# B&R Automation Studio project NAEUL004C00R13L518F00 (part 27)

#### Act_OptP1031TravMask.st
```iecst
ACTION Act_OptP1031TravMask:

	// Interlock Power
	IF p_bTravAxisErr = TRUE AND p_bTravPwrOn = FALSE THEN
		fUIInRtStatOff(ADR(tyP1031MagSetTeach.tyMotionStdTrav.tyBtnPwr.uiMaskRtStat));
		tyP1031MagSetTeach.tyMotionStdTrav.tyBtnPwr.bValue		:= FALSE;
	ELSE
		fUIInRtStatHide(ADR(tyP1031MagSetTeach.tyMotionStdTrav.tyBtnPwr.uiMaskRtStat));
	END_IF

	// Interlock Others Move
	IF p_bTravAxisErr = TRUE OR p_bTravPwrOn = FALSE THEN
		fUIInRtStatOff(ADR(tyP1031MagSetTeach.tyMotionStdTrav.tyBtnOrigin.uiMaskRtStat));
		fUIInRtStatOff(ADR(tyP1031MagSetTeach.tyMotionStdTrav.tyBtnMovRel.uiMaskRtStat));
		fUIInRtStatOff(ADR(tyP1031MagSetTeach.tyMotionStdTrav.tyBtnJogFront.uiMaskRtStat));
		fUIInRtStatOff(ADR(tyP1031MagSetTeach.tyMotionStdTrav.tyBtnJogRear.uiMaskRtStat));
	ELSE
		fUIInRtStatHide(ADR(tyP1031MagSetTeach.tyMotionStdTrav.tyBtnOrigin.uiMaskRtStat));
		fUIInRtStatHide(ADR(tyP1031MagSetTeach.tyMotionStdTrav.tyBtnMovRel.uiMaskRtStat));
		fUIInRtStatHide(ADR(tyP1031MagSetTeach.tyMotionStdTrav.tyBtnJogFront.uiMaskRtStat));
		fUIInRtStatHide(ADR(tyP1031MagSetTeach.tyMotionStdTrav.tyBtnJogRear.uiMaskRtStat));
	END_IF

	// Interlock Move Absolute
	IF p_bTravAxisErr = TRUE OR p_bTravPwrOn = FALSE OR p_bTravIsHomed = FALSE THEN
		fUIInRtStatOff(ADR(tyP1031MagSetTeach.tyTeachTravPosMag1.tyBtn2.uiMaskRtStat));
		fUIInRtStatOff(ADR(tyP1031MagSetTeach.tyTeachTravPosMag2.tyBtn2.uiMaskRtStat));
		fUIInRtStatOff(ADR(tyP1031MagSetTeach.tyTeachTravPosMag3.tyBtn2.uiMaskRtStat));
		fUIInRtStatOff(ADR(tyP1031MagSetTeach.tyMotionStdTrav.tyBtnMovAbs.uiMaskRtStat));
	ELSE
		fUIInRtStatHide(ADR(tyP1031MagSetTeach.tyTeachTravPosMag1.tyBtn2.uiMaskRtStat));
		fUIInRtStatHide(ADR(tyP1031MagSetTeach.tyTeachTravPosMag2.tyBtn2.uiMaskRtStat));
		fUIInRtStatHide(ADR(tyP1031MagSetTeach.tyTeachTravPosMag3.tyBtn2.uiMaskRtStat));
		fUIInRtStatHide(ADR(tyP1031MagSetTeach.tyMotionStdTrav.tyBtnMovAbs.uiMaskRtStat));
	END_IF

	//Interlock Limit Sensor
	IF tyP1031MagSetTeach.tyMotionStdTrav.tyBtnRearLmtSen.bValue = TRUE THEN
		fUIInRtStatOff(ADR(tyP1031MagSetTeach.tyMotionStdTrav.tyBtnJogRear.uiMaskRtStat));
	END_IF

	IF tyP1031MagSetTeach.tyMotionStdTrav.tyBtnFrontLmtSen.bValue = TRUE THEN
		fUIInRtStatOff(ADR(tyP1031MagSetTeach.tyMotionStdTrav.tyBtnJogFront.uiMaskRtStat));
	END_IF

	// Interlock When Moving
	IF tyP1031MagSetTeach.tyMotionStdTrav.tyBtnOrigin.bRtCompl = TRUE THEN
		fUIInRtStatOff(ADR(tyP1031MagSetTeach.tyMotionStdTrav.tyBtnMovAbs.uiMaskRtStat));
		fUIInRtStatOff(ADR(tyP1031MagSetTeach.tyMotionStdTrav.tyBtnMovRel.uiMaskRtStat));
		fUIInRtStatOff(ADR(tyP1031MagSetTeach.tyMotionStdTrav.tyBtnJogFront.uiMaskRtStat));
		fUIInRtStatOff(ADR(tyP1031MagSetTeach.tyMotionStdTrav.tyBtnJogRear.uiMaskRtStat));

		fUIInRtStatOff(ADR(tyP1031MagSetTeach.tyTeachTravPosMag1.tyBtn2.uiMaskRtStat));
		fUIInRtStatOff(ADR(tyP1031MagSetTeach.tyTeachTravPosMag2.tyBtn2.uiMaskRtStat));
		fUIInRtStatOff(ADR(tyP1031MagSetTeach.tyTeachTravPosMag3.tyBtn2.uiMaskRtStat));

	ELSIF tyP1031MagSetTeach.tyMotionStdTrav.tyBtnMovAbs.bRtCompl = TRUE THEN
		fUIInRtStatOff(ADR(tyP1031MagSetTeach.tyMotionStdTrav.tyBtnOrigin.uiMaskRtStat));
		fUIInRtStatOff(ADR(tyP1031MagSetTeach.tyMotionStdTrav.tyBtnMovRel.uiMaskRtStat));
		fUIInRtStatOff(ADR(tyP1031MagSetTeach.tyMotionStdTrav.tyBtnJogFront.uiMaskRtStat));
		fUIInRtStatOff(ADR(tyP1031MagSetTeach.tyMotionStdTrav.tyBtnJogRear.uiMaskRtStat));

		fUIInRtStatOff(ADR(tyP1031MagSetTeach.tyTeachTravPosMag1.tyBtn2.uiMaskRtStat));
		fUIInRtStatOff(ADR(tyP1031MagSetTeach.tyTeachTravPosMag2.tyBtn2.uiMaskRtStat));
		fUIInRtStatOff(ADR(tyP1031MagSetTeach.tyTeachTravPosMag3.tyBtn2.uiMaskRtStat));

	ELSIF tyP1031MagSetTeach.tyMotionStdTrav.tyBtnMovRel.bRtCompl = TRUE THEN
		fUIInRtStatOff(ADR(tyP1031MagSetTeach.tyMotionStdTrav.tyBtnOrigin.uiMaskRtStat));
		fUIInRtStatOff(ADR(tyP1031MagSetTeach.tyMotionStdTrav.tyBtnMovAbs.uiMaskRtStat));
		fUIInRtStatOff(ADR(tyP1031MagSetTeach.tyMotionStdTrav.tyBtnJogFront.uiMaskRtStat));
		fUIInRtStatOff(ADR(tyP1031MagSetTeach.tyMotionStdTrav.tyBtnJogRear.uiMaskRtStat));

		fUIInRtStatOff(ADR(tyP1031MagSetTeach.tyTeachTravPosMag1.tyBtn2.uiMaskRtStat));
		fUIInRtStatOff(ADR(tyP1031MagSetTeach.tyTeachTravPosMag2.tyBtn2.uiMaskRtStat));
		fUIInRtStatOff(ADR(tyP1031MagSetTeach.tyTeachTravPosMag3.tyBtn2.uiMaskRtStat));

	ELSIF tyP1031MagSetTeach.tyMotionStdTrav.tyBtnJogRear.bRtCompl = TRUE OR tyP1031MagSetTeach.tyMotionStdTrav.tyBtnJogRear.bValue = TRUE THEN
		fUIInRtStatOff(ADR(tyP1031MagSetTeach.tyMotionStdTrav.tyBtnOrigin.uiMaskRtStat));
		fUIInRtStatOff(ADR(tyP1031MagSetTeach.tyMotionStdTrav.tyBtnMovAbs.uiMaskRtStat));
		fUIInRtStatOff(ADR(tyP1031MagSetTeach.tyMotionStdTrav.tyBtnMovRel.uiMaskRtStat));
		fUIInRtStatOff(ADR(tyP1031MagSetTeach.tyMotionStdTrav.tyBtnJogFront.uiMaskRtStat));

		fUIInRtStatOff(ADR(tyP1031MagSetTeach.tyTeachTravPosMag1.tyBtn2.uiMaskRtStat));
		fUIInRtStatOff(ADR(tyP1031MagSetTeach.tyTeachTravPosMag2.tyBtn2.uiMaskRtStat));
		fUIInRtStatOff(ADR(tyP1031MagSetTeach.tyTeachTravPosMag3.tyBtn2.uiMaskRtStat));

	ELSIF tyP1031MagSetTeach.tyMotionStdTrav.tyBtnJogFront.bRtCompl = TRUE OR tyP1031MagSetTeach.tyMotionStdTrav.tyBtnJogFront.bValue = TRUE THEN
		fUIInRtStatOff(ADR(tyP1031MagSetTeach.tyMotionStdTrav.tyBtnOrigin.uiMaskRtStat));
		fUIInRtStatOff(ADR(tyP1031MagSetTeach.tyMotionStdTrav.tyBtnMovAbs.uiMaskRtStat));
		fUIInRtStatOff(ADR(tyP1031MagSetTeach.tyMotionStdTrav.tyBtnMovRel.uiMaskRtStat));
		fUIInRtStatOff(ADR(tyP1031MagSetTeach.tyMotionStdTrav.tyBtnJogRear.uiMaskRtStat));

		fUIInRtStatOff(ADR(tyP1031MagSetTeach.tyTeachTravPosMag1.tyBtn2.uiMaskRtStat));
		fUIInRtStatOff(ADR(tyP1031MagSetTeach.tyTeachTravPosMag2.tyBtn2.uiMaskRtStat));
		fUIInRtStatOff(ADR(tyP1031MagSetTeach.tyTeachTravPosMag3.tyBtn2.uiMaskRtStat));

	ELSIF tyP1031MagSetTeach.tyTeachTravPosMag1.tyBtn2.bRtCompl = TRUE THEN
		fUIInRtStatOff(ADR(tyP1031MagSetTeach.tyMotionStdTrav.tyBtnOrigin.uiMaskRtStat));
		fUIInRtStatOff(ADR(tyP1031MagSetTeach.tyMotionStdTrav.tyBtnMovAbs.uiMaskRtStat));
		fUIInRtStatOff(ADR(tyP1031MagSetTeach.tyMotionStdTrav.tyBtnMovRel.uiMaskRtStat));
		fUIInRtStatOff(ADR(tyP1031MagSetTeach.tyMotionStdTrav.tyBtnJogFront.uiMaskRtStat));
		fUIInRtStatOff(ADR(tyP1031MagSetTeach.tyMotionStdTrav.tyBtnJogRear.uiMaskRtStat));

	ELSIF tyP1031MagSetTeach.tyTeachTravPosMag2.tyBtn2.bRtCompl = TRUE THEN
		fUIInRtStatOff(ADR(tyP1031MagSetTeach.tyMotionStdTrav.tyBtnOrigin.uiMaskRtStat));
		fUIInRtStatOff(ADR(tyP1031MagSetTeach.tyMotionStdTrav.tyBtnMovAbs.uiMaskRtStat));
		fUIInRtStatOff(ADR(tyP1031MagSetTeach.tyMotionStdTrav.tyBtnMovRel.uiMaskRtStat));
		fUIInRtStatOff(ADR(tyP1031MagSetTeach.tyMotionStdTrav.tyBtnJogFront.uiMaskRtStat));
		fUIInRtStatOff(ADR(tyP1031MagSetTeach.tyMotionStdTrav.tyBtnJogRear.uiMaskRtStat));

	ELSIF tyP1031MagSetTeach.tyTeachTravPosMag3.tyBtn2.bRtCompl = TRUE THEN
		fUIInRtStatOff(ADR(tyP1031MagSetTeach.tyMotionStdTrav.tyBtnOrigin.uiMaskRtStat));
		fUIInRtStatOff(ADR(tyP1031MagSetTeach.tyMotionStdTrav.tyBtnMovAbs.uiMaskRtStat));
		fUIInRtStatOff(ADR(tyP1031MagSetTeach.tyMotionStdTrav.tyBtnMovRel.uiMaskRtStat));
		fUIInRtStatOff(ADR(tyP1031MagSetTeach.tyMotionStdTrav.tyBtnJogFront.uiMaskRtStat));
		fUIInRtStatOff(ADR(tyP1031MagSetTeach.tyMotionStdTrav.tyBtnJogRear.uiMaskRtStat));

	END_IF

	//Axis Error
	IF tyP1031MagSetTeach.tyMotionStdTrav.tyBtnPwr.bRtCompl = TRUE  THEN
		fUIInRtStatOff(ADR(tyP1031MagSetTeach.tyMotionStdTrav.tyBtnRst.uiMaskRtStat));
	ELSE
		fUIInRtStatHide(ADR(tyP1031MagSetTeach.tyMotionStdTrav.tyBtnRst.uiMaskRtStat));
	END_IF

	//Interlock Button Get
	IF p_bTravAxisErr = TRUE OR p_bTravIsHomed = FALSE OR p_bTravFwdLmtSen = TRUE OR p_bTravRevLmtSen = TRUE THEN
		fUIInRtStatOff(ADR(tyP1031MagSetTeach.tyTeachTravPosMag1.tyBtn1.uiMaskRtStat));
		fUIInRtStatOff(ADR(tyP1031MagSetTeach.tyTeachTravPosMag2.tyBtn1.uiMaskRtStat));
		fUIInRtStatOff(ADR(tyP1031MagSetTeach.tyTeachTravPosMag3.tyBtn1.uiMaskRtStat));
	ELSE
		fUIInRtStatHide(ADR(tyP1031MagSetTeach.tyTeachTravPosMag1.tyBtn1.uiMaskRtStat));
		fUIInRtStatHide(ADR(tyP1031MagSetTeach.tyTeachTravPosMag2.tyBtn1.uiMaskRtStat));
		fUIInRtStatHide(ADR(tyP1031MagSetTeach.tyTeachTravPosMag3.tyBtn1.uiMaskRtStat));
	END_IF

END_ACTION
```

#### Act_OptP1031TravUpdtDat.st
```iecst
ACTION Act_OptP1031TravUpdtDat:

	tyP1031MagSetTeach.tyMotionStdTrav.tyNumCurrPos.diValue			:= p_diTravActualPos;
	tyP1031MagSetTeach.tyMotionStdTrav.tyNumErrCode.diValue			:= UDINT_TO_DINT(p_udiTravAxisErrID);
	tyP1031MagSetTeach.tyMotionStdTrav.tyBitmapPwr.usiValueIdx		:= BOOL_TO_USINT(p_bTravPwrOn);
	tyP1031MagSetTeach.tyMotionStdTrav.tyBitmapRst.usiValueIdx		:= BOOL_TO_USINT(NOT p_bTravAxisErr);
	tyP1031MagSetTeach.tyMotionStdTrav.tyBitmapOrigin.usiValueIdx	:= BOOL_TO_USINT(p_bTravIsHomed);
	tyP1031MagSetTeach.tyMotionStdTrav.tyBtnFrontLmtSen.bValue		:= p_bTravFrontSen;
	tyP1031MagSetTeach.tyMotionStdTrav.tyBtnRearLmtSen.bValue		:= p_bTravRearSen;

	//Machine Bitmap
	IF p_bTravIsHomed = TRUE THEN
		IF p_diTravActualPos <= (p_tyNtParamCurr.tyUITravTargetPos.diMax / 3) THEN
			tyP1031MagSetTeach.tyMotionStdTrav.tyBitmapMc.uiValueIdx 	:= 5;
		ELSIF p_diTravActualPos <= (p_tyNtParamCurr.tyUITravTargetPos.diMax / 3 * 2) THEN
			tyP1031MagSetTeach.tyMotionStdTrav.tyBitmapMc.uiValueIdx 	:= 6;
		ELSE
			tyP1031MagSetTeach.tyMotionStdTrav.tyBitmapMc.uiValueIdx 	:= 7;
		END_IF
	ELSE
		tyP1031MagSetTeach.tyMotionStdTrav.tyBitmapMc.uiValueIdx	:= 5;
	END_IF

	IF p_tyNtParamCurr.eProjMag = ULMagDual THEN
		IF p_tyNtParamCurr.bProjLifterMagPlatform AND p_tyNtParamCurr.bUIConvDirRL THEN
			IF 	tyP1031MagSetTeach.tyMotionStdTrav.tyBitmapMc.uiValueIdx < 700 THEN
				tyP1031MagSetTeach.tyMotionStdTrav.tyBitmapMc.uiValueIdx	:= tyP1031MagSetTeach.tyMotionStdTrav.tyBitmapMc.uiValueIdx + 700;
			END_IF
		ELSIF p_tyNtParamCurr.bProjLifterMagPlatform THEN
			IF 	tyP1031MagSetTeach.tyMotionStdTrav.tyBitmapMc.uiValueIdx < 600 THEN
				tyP1031MagSetTeach.tyMotionStdTrav.tyBitmapMc.uiValueIdx	:= tyP1031MagSetTeach.tyMotionStdTrav.tyBitmapMc.uiValueIdx + 600;
			END_IF
		ELSIF p_tyNtParamCurr.bMagAutoVerifyPrep = FALSE THEN
			IF 	tyP1031MagSetTeach.tyMotionStdTrav.tyBitmapMc.uiValueIdx < 100 THEN
				tyP1031MagSetTeach.tyMotionStdTrav.tyBitmapMc.uiValueIdx	:= tyP1031MagSetTeach.tyMotionStdTrav.tyBitmapMc.uiValueIdx + 300;
			END_IF
		ELSE
			IF 	tyP1031MagSetTeach.tyMotionStdTrav.tyBitmapMc.uiValueIdx < 300 THEN
				tyP1031MagSetTeach.tyMotionStdTrav.tyBitmapMc.uiValueIdx	:= tyP1031MagSetTeach.tyMotionStdTrav.tyBitmapMc.uiValueIdx + 300;
			END_IF
		END_IF
	ELSIF p_tyNtParamCurr.eProjMag = ULMagTriple THEN
		IF p_tyNtParamCurr.bProjLifterMagPlatform AND p_tyNtParamCurr.bUIConvDirRL THEN
			IF 	tyP1031MagSetTeach.tyMotionStdTrav.tyBitmapMc.uiValueIdx < 800 THEN
				tyP1031MagSetTeach.tyMotionStdTrav.tyBitmapMc.uiValueIdx	:= tyP1031MagSetTeach.tyMotionStdTrav.tyBitmapMc.uiValueIdx + 800;
			END_IF
		ELSIF p_tyNtParamCurr.bProjLifterMagPlatform THEN
			IF 	tyP1031MagSetTeach.tyMotionStdTrav.tyBitmapMc.uiValueIdx < 500 THEN
				tyP1031MagSetTeach.tyMotionStdTrav.tyBitmapMc.uiValueIdx	:= tyP1031MagSetTeach.tyMotionStdTrav.tyBitmapMc.uiValueIdx + 500;
			END_IF
		ELSIF p_tyNtParamCurr.bMagAutoVerifyPrep = TRUE AND p_tyNtParamCurr.bProjMotorizedPusherPrep = FALSE THEN
			IF 	tyP1031MagSetTeach.tyMotionStdTrav.tyBitmapMc.uiValueIdx < 200 THEN
				tyP1031MagSetTeach.tyMotionStdTrav.tyBitmapMc.uiValueIdx	:= tyP1031MagSetTeach.tyMotionStdTrav.tyBitmapMc.uiValueIdx + 200;
			END_IF
		ELSIF p_tyNtParamCurr.bMagAutoVerifyPrep = FALSE AND p_tyNtParamCurr.bProjMotorizedPusherPrep = TRUE THEN
			IF 	tyP1031MagSetTeach.tyMotionStdTrav.tyBitmapMc.uiValueIdx < 400 THEN
				tyP1031MagSetTeach.tyMotionStdTrav.tyBitmapMc.uiValueIdx	:= tyP1031MagSetTeach.tyMotionStdTrav.tyBitmapMc.uiValueIdx + 400;
			END_IF
		END_IF
	END_IF

END_ACTION
```

#### Act_OptP1031TravKeypad.st
```iecst
ACTION Act_OptP1031TravKeypad:

	IF fUIOutRtStatTPIsOpen(ADR(tyP1031MagSetTeach.tyMotionStdTrav.tyNumTargetPos.uiRtStat)) = TRUE THEN
		tyProperty.tyKeypad.tyStringTitle.sKeypadTitle		:= tyP1031MagSetTeach.tyMotionStdTrav.tyNumTargetPos.sKeypadTitle;

	ELSIF fUIOutRtStatTPIsOpen(ADR(tyP1031MagSetTeach.tyMotionStdTrav.tyNumStepSize.uiRtStat)) = TRUE THEN
		tyProperty.tyKeypad.tyStringTitle.sKeypadTitle		:= tyP1031MagSetTeach.tyMotionStdTrav.tyNumStepSize.sKeypadTitle;

	ELSIF fUIOutRtStatTPIsOpen(ADR(tyP1031MagSetTeach.tyMotionStdTrav.tyNumNomSpd.uiRtStat)) = TRUE THEN
		tyProperty.tyKeypad.tyStringTitle.sKeypadTitle		:= tyP1031MagSetTeach.tyMotionStdTrav.tyNumNomSpd.sKeypadTitle;

	ELSIF fUIOutRtStatTPIsOpen(ADR(tyP1031MagSetTeach.tyMotionStdTrav.tyNumSlwSpd.uiRtStat)) = TRUE THEN
		tyProperty.tyKeypad.tyStringTitle.sKeypadTitle		:= tyP1031MagSetTeach.tyMotionStdTrav.tyNumSlwSpd.sKeypadTitle;
	END_IF

END_ACTION
```

#### Act_OptP1031TravRstMnl.st
```iecst
ACTION Act_OptP1031TravRstMnl:

	IF EDGEPOS((bManualMod = FALSE) OR (p_eTravStatus = Error)) THEN

		bJogSlow				:= FALSE;
		bJogFast				:= FALSE;
		fbJogSlowToFastDlyTm.IN	:= FALSE;

		tyP1031MagSetTeach.tyMotionStdTrav.tyBtnPwr.bRtCompl			:= FALSE;
		tyP1031MagSetTeach.tyMotionStdTrav.tyBtnStop.bRtCompl			:= FALSE;
		tyP1031MagSetTeach.tyMotionStdTrav.tyBtnOrigin.bRtCompl			:= FALSE;
		tyP1031MagSetTeach.tyMotionStdTrav.tyBtnRst.bRtCompl			:= FALSE;
		tyP1031MagSetTeach.tyMotionStdTrav.tyBtnMovAbs.bRtCompl			:= FALSE;
		tyP1031MagSetTeach.tyMotionStdTrav.tyBtnMovRel.bRtCompl			:= FALSE;
		tyP1031MagSetTeach.tyMotionStdTrav.tyBtnJogFront.bRtCompl		:= FALSE;
		tyP1031MagSetTeach.tyMotionStdTrav.tyBtnJogRear.bRtCompl		:= FALSE;

		tyP1031MagSetTeach.tyTeachTravPosMag1.tyBtn2.bRtCompl			:= FALSE;
		tyP1031MagSetTeach.tyTeachTravPosMag2.tyBtn2.bRtCompl			:= FALSE;
		tyP1031MagSetTeach.tyTeachTravPosMag3.tyBtn2.bRtCompl			:= FALSE;

		tyP1031MagSetTeach.tyMotionStdTrav.tyBtnPwr.bValue				:= FALSE;
		tyP1031MagSetTeach.tyMotionStdTrav.tyBtnStop.bValue				:= TRUE;
		tyP1031MagSetTeach.tyMotionStdTrav.tyBtnOrigin.bValue			:= FALSE;
		tyP1031MagSetTeach.tyMotionStdTrav.tyBtnRst.bValue				:= FALSE;
		tyP1031MagSetTeach.tyMotionStdTrav.tyBtnMovAbs.bValue			:= FALSE;
		tyP1031MagSetTeach.tyMotionStdTrav.tyBtnMovRel.bValue			:= FALSE;
		tyP1031MagSetTeach.tyMotionStdTrav.tyBtnJogFront.bValue			:= FALSE;
		tyP1031MagSetTeach.tyMotionStdTrav.tyBtnJogRear.bValue			:= FALSE;

		tyP1031MagSetTeach.tyTeachTravPosMag1.tyBtn2.bValue				:= FALSE;
		tyP1031MagSetTeach.tyTeachTravPosMag2.tyBtn2.bValue				:= FALSE;
		tyP1031MagSetTeach.tyTeachTravPosMag3.tyBtn2.bValue				:= FALSE;

		tyP1031MagSetTeach.tyMotionStdTrav.tyBtnPwr.bRtLk				:= FALSE;
		tyP1031MagSetTeach.tyMotionStdTrav.tyBtnStop.bRtLk				:= TRUE;
		tyP1031MagSetTeach.tyMotionStdTrav.tyBtnOrigin.bRtLk			:= FALSE;
		tyP1031MagSetTeach.tyMotionStdTrav.tyBtnRst.bRtLk				:= FALSE;
		tyP1031MagSetTeach.tyMotionStdTrav.tyBtnMovAbs.bRtLk			:= FALSE;
		tyP1031MagSetTeach.tyMotionStdTrav.tyBtnMovRel.bRtLk			:= FALSE;
		tyP1031MagSetTeach.tyMotionStdTrav.tyBtnJogFront.bRtLk			:= FALSE;
		tyP1031MagSetTeach.tyMotionStdTrav.tyBtnJogRear.bRtLk			:= FALSE;

		tyP1031MagSetTeach.tyTeachTravPosMag1.tyBtn2.bRtLk				:= FALSE;
		tyP1031MagSetTeach.tyTeachTravPosMag2.tyBtn2.bRtLk				:= FALSE;
		tyP1031MagSetTeach.tyTeachTravPosMag3.tyBtn2.bRtLk				:= FALSE;

		tyP1031MagSetTeach.tyMotionStdTrav.tyBtnPwr.uiMaskRtStat		:= TRUE;
		tyP1031MagSetTeach.tyMotionStdTrav.tyBtnOrigin.uiMaskRtStat		:= FALSE;
		tyP1031MagSetTeach.tyMotionStdTrav.tyBtnRst.uiMaskRtStat		:= TRUE;
		tyP1031MagSetTeach.tyMotionStdTrav.tyBtnMovAbs.uiMaskRtStat		:= FALSE;
		tyP1031MagSetTeach.tyMotionStdTrav.tyBtnMovRel.uiMaskRtStat		:= FALSE;
		tyP1031MagSetTeach.tyMotionStdTrav.tyBtnJogFront.uiMaskRtStat	:= FALSE;
		tyP1031MagSetTeach.tyMotionStdTrav.tyBtnJogRear.uiMaskRtStat	:= FALSE;

		tyP1031MagSetTeach.tyTeachTravPosMag1.tyBtn2.uiMaskRtStat		:= FALSE;
		tyP1031MagSetTeach.tyTeachTravPosMag2.tyBtn2.uiMaskRtStat		:= FALSE;
		tyP1031MagSetTeach.tyTeachTravPosMag3.tyBtn2.uiMaskRtStat		:= FALSE;

		eInShutterAct	:= PneuActIdle;
		eOutShutterAct	:= PneuActIdle;
		eOutShutterAct2	:= PneuActIdle;
		eOutShutterAct3	:= PneuActIdle;
		eTravAct	:= TravActIdle;

		tyP1031MagSetTeach.tyInOutletShutterFB.tyBtnClose.bRtCompl	:= FALSE;
		tyP1031MagSetTeach.tyInOutletShutterFB.tyBtnClose.bValue	:= FALSE;
		tyP1031MagSetTeach.tyInOutletShutterFB.tyBtnOpen.bRtCompl	:= FALSE;
		tyP1031MagSetTeach.tyInOutletShutterFB.tyBtnOpen.bValue	:= FALSE;

	END_IF

END_ACTION
```

#### Act_OptP1031LifterTeach.st
```iecst
ACTION Act_OptP1031LifterTeach:

	IF tyP1031MagSetTeach.tyTeachLifterMag1Slt1Pos.tyBtn1.bRtCompl = TRUE THEN // Teach Lifter Magazine 1 Slot 1 Position

		p_tyC0008MsgBox ACCESS ADR(tyP1031MagSetTeach.tyMsgBoxUpdtLifterMag1Slt1Pos);

		IF tyP1031MagSetTeach.tyMsgBoxUpdtLifterMag1Slt1Pos.tyBtnNo.bRtCompl THEN
			tyP1031MagSetTeach.tyMsgBoxUpdtLifterMag1Slt1Pos.tyBtnNo.bRtCompl 	:= FALSE;
			tyP1031MagSetTeach.tyMsgBoxUpdtLifterMag1Slt1Pos.tyBtnNo.bValue 	:= FALSE;

			p_tyC0008MsgBox ACCESS ADR(tyP1031MagSetTeach.tyMsgBoxHide);

			//Write Actual Position To Magazine Setting.
			tyP1030MagSet.tyMagSet.tyNumLifterMag1Slt1Pos.diValue 	:= p_diLifterBtmActualPos;
			tyP1030MagSet.tyMagSet.tyNumLifterMag1Slt1Pos.bRtCompl	:= TRUE;

			//Back To Magazine Settings
			eChgPage	:= UIP1030MagSet;

			fUIInRtStatHide(ADR(tyP1030MagSet.tyMagSet.tyBtnSave.uiMaskRtStat));

			tyP1031MagSetTeach.tyTeachLifterMag1Slt1Pos.tyBtn1.bRtCompl	:= FALSE;
			tyP1031MagSetTeach.tyTeachLifterMag1Slt1Pos.tyBtn1.bValue	:= FALSE;

		END_IF

	ELSIF tyP1031MagSetTeach.tyTeachLifterMag2Slt1Pos.tyBtn1.bRtCompl = TRUE THEN // Teach Lifter Magazine 2 Slot 1 Position

		p_tyC0008MsgBox ACCESS ADR(tyP1031MagSetTeach.tyMsgBoxUpdtLifterMag2Slt1Pos);

		IF tyP1031MagSetTeach.tyMsgBoxUpdtLifterMag2Slt1Pos.tyBtnNo.bRtCompl THEN
			tyP1031MagSetTeach.tyMsgBoxUpdtLifterMag2Slt1Pos.tyBtnNo.bRtCompl 	:= FALSE;
			tyP1031MagSetTeach.tyMsgBoxUpdtLifterMag2Slt1Pos.tyBtnNo.bValue 	:= FALSE;

			p_tyC0008MsgBox ACCESS ADR(tyP1031MagSetTeach.tyMsgBoxHide);

			IF p_tyNtParamCurr.bProjMagConvLane2Prep THEN
				tyP1030MagSet.tyMagSet.tyNumLifterMag2Slt1Pos.diValue 	:= p_diLifter2ActualPos;
			ELSE
				//Write Actual Position To Magazine Setting.
				tyP1030MagSet.tyMagSet.tyNumLifterMag2Slt1Pos.diValue 	:= p_diLifterBtmActualPos;
			END_IF

			tyP1030MagSet.tyMagSet.tyNumLifterMag2Slt1Pos.bRtCompl	:= TRUE;

			//Back To Magazine Settings
			eChgPage	:= UIP1030MagSet;

			fUIInRtStatHide(ADR(tyP1030MagSet.tyMagSet.tyBtnSave.uiMaskRtStat));

			tyP1031MagSetTeach.tyTeachLifterMag2Slt1Pos.tyBtn1.bRtCompl	:= FALSE;
			tyP1031MagSetTeach.tyTeachLifterMag2Slt1Pos.tyBtn1.bValue	:= FALSE;

		END_IF

	ELSIF tyP1031MagSetTeach.tyTeachLifterMag3Slt1Pos.tyBtn1.bRtCompl = TRUE THEN // Teach Lifter Magazine 3 Slot 1 Position

		p_tyC0008MsgBox ACCESS ADR(tyP1031MagSetTeach.tyMsgBoxUpdtLifterMag3Slt1Pos);

		IF tyP1031MagSetTeach.tyMsgBoxUpdtLifterMag3Slt1Pos.tyBtnNo.bRtCompl THEN
			tyP1031MagSetTeach.tyMsgBoxUpdtLifterMag3Slt1Pos.tyBtnNo.bRtCompl 	:= FALSE;
			tyP1031MagSetTeach.tyMsgBoxUpdtLifterMag3Slt1Pos.tyBtnNo.bValue 	:= FALSE;

			p_tyC0008MsgBox ACCESS ADR(tyP1031MagSetTeach.tyMsgBoxHide);

			//Write Actual Position To Magazine Setting.
			tyP1030MagSet.tyMagSet.tyNumLifterMag3Slt1Pos.diValue 	:= p_diLifterBtmActualPos;
			tyP1030MagSet.tyMagSet.tyNumLifterMag3Slt1Pos.bRtCompl	:= TRUE;

			//Back To Magazine Settings
			eChgPage	:= UIP1030MagSet;

			fUIInRtStatHide(ADR(tyP1030MagSet.tyMagSet.tyBtnSave.uiMaskRtStat));

			tyP1031MagSetTeach.tyTeachLifterMag3Slt1Pos.tyBtn1.bRtCompl	:= FALSE;
			tyP1031MagSetTeach.tyTeachLifterMag3Slt1Pos.tyBtn1.bValue	:= FALSE;

		END_IF

	END_IF

END_ACTION
```

#### Act_OptP1031LifterFBCtrl.st
```iecst
ACTION Act_OptP1031LifterFBCtrl:

	fbJogSlowToFastDlyTm.PT	:= T#2s;
	fbJogSlowToFastDlyTm;
	fbLmtRstTm;

	//Lifter Safety Sensor Interruption
	IF EDGENEG(p_tyDI.bLifterSafetyLmtSW1 AND p_tyDI.bLifterSafetyLmtSW2 AND p_tyDI.bLifterTimingBeltSen) THEN
		tyP1031MagSetTeach.tyMotionStdLifter.tyBtnStop.bRtCompl	:= TRUE;
	END_IF

//	IF EDGEPOS((p_udiLifterBtmAxisErrID = 21570 OR p_udiLifterBtmAxisErrID = 21571) AND tyP1031MagSetTeach.tyMotionStdLifter.tyBtnJogDown.bValue = FALSE AND tyP1031MagSetTeach.tyMotionStdLifter.tyBtnJogUp.bValue = FALSE) THEN
	IF EDGEPOS((p_bLifterBtmFwdLmtSen OR p_bLifterBtmRevLmtSen OR p_udiLifterBtmAxisErrID = 21570 OR p_udiLifterBtmAxisErrID = 21571)
		AND tyP1026McSetTeach.tyMotionStdLifter.tyBtnJogDown.bValue = FALSE
		AND tyP1026McSetTeach.tyMotionStdLifter.tyBtnJogUp.bValue = FALSE) THEN
			fbLmtRstTm.IN				:= TRUE;
	END_IF

	IF fbLmtRstTm.Q = TRUE THEN
		tyP1031MagSetTeach.tyMotionStdLifter.tyBtnRst.bRtCompl		:= TRUE;
	END_IF

	IF (tyP1031MagSetTeach.tyMotionStdLifter.tyBtnJogUp.bValue = FALSE AND tyP1031MagSetTeach.tyMotionStdLifter.tyBtnJogDown.bValue = FALSE) AND (p_bLifterBtmJogging = TRUE) THEN
		bJogStopLifter	:= TRUE;
	END_IF

	IF tyP1031MagSetTeach.tyMotionStdLifter.tyBtnStop.bRtCompl = TRUE THEN
		eLifterBtmAct		:= LifterActStop;

		IF p_eLifterBtmStat = LifterActStop AND p_eLifterBtmStatus = Done THEN
			eLifterBtmAct	:= LifterActIdle;

			tyP1031MagSetTeach.tyMotionStdLifter.tyBtnStop.bRtCompl			:= FALSE;
			tyP1031MagSetTeach.tyMotionStdLifter.tyBtnJogDown.bRtCompl		:= FALSE;
			tyP1031MagSetTeach.tyMotionStdLifter.tyBtnJogUp.bRtCompl		:= FALSE;
			tyP1031MagSetTeach.tyMotionStdLifter.tyBtnOrigin.bRtCompl		:= FALSE;
			tyP1031MagSetTeach.tyMotionStdLifter.tyBtnMovAbs.bRtCompl		:= FALSE;
			tyP1031MagSetTeach.tyMotionStdLifter.tyBtnMovRel.bRtCompl		:= FALSE;

			tyP1031MagSetTeach.tyTeachLifterMag1Slt1Pos.tyBtn2.bRtCompl		:= FALSE;
			tyP1031MagSetTeach.tyTeachLifterMag2Slt1Pos.tyBtn2.bRtCompl		:= FALSE;
			tyP1031MagSetTeach.tyTeachLifterMag3Slt1Pos.tyBtn2.bRtCompl		:= FALSE;

			tyP1031MagSetTeach.tyMotionStdLifter.tyBtnStop.bValue			:= TRUE;
			tyP1031MagSetTeach.tyMotionStdLifter.tyBtnJogDown.bValue		:= FALSE;
			tyP1031MagSetTeach.tyMotionStdLifter.tyBtnJogUp.bValue			:= FALSE;
			tyP1031MagSetTeach.tyMotionStdLifter.tyBtnOrigin.bValue			:= FALSE;
			tyP1031MagSetTeach.tyMotionStdLifter.tyBtnMovAbs.bValue			:= FALSE;
			tyP1031MagSetTeach.tyMotionStdLifter.tyBtnMovRel.bValue			:= FALSE;

			tyP1031MagSetTeach.tyTeachLifterMag1Slt1Pos.tyBtn2.bValue		:= FALSE;
			tyP1031MagSetTeach.tyTeachLifterMag2Slt1Pos.tyBtn2.bValue		:= FALSE;
			tyP1031MagSetTeach.tyTeachLifterMag3Slt1Pos.tyBtn2.bValue		:= FALSE;

			tyP1031MagSetTeach.tyMotionStdLifter.tyBtnStop.bRtLk			:= TRUE;
			tyP1031MagSetTeach.tyMotionStdLifter.tyBtnJogDown.bRtLk			:= FALSE;
			tyP1031MagSetTeach.tyMotionStdLifter.tyBtnJogUp.bRtLk			:= FALSE;
			tyP1031MagSetTeach.tyMotionStdLifter.tyBtnOrigin.bRtLk			:= FALSE;
			tyP1031MagSetTeach.tyMotionStdLifter.tyBtnMovAbs.bRtLk			:= FALSE;
			tyP1031MagSetTeach.tyMotionStdLifter.tyBtnMovRel.bRtLk			:= FALSE;

			tyP1031MagSetTeach.tyTeachLifterMag1Slt1Pos.tyBtn2.bRtLk		:= FALSE;
			tyP1031MagSetTeach.tyTeachLifterMag2Slt1Pos.tyBtn2.bRtLk		:= FALSE;
			tyP1031MagSetTeach.tyTeachLifterMag3Slt1Pos.tyBtn2.bRtLk		:= FALSE;

		END_IF

	ELSIF (tyP1031MagSetTeach.tyMotionStdLifter.tyBtnJogDown.bRtCompl = TRUE) OR (tyP1031MagSetTeach.tyMotionStdLifter.tyBtnJogUp.bRtCompl = TRUE) OR (bJogStopLifter = TRUE) THEN
		bJogSlow					:= FALSE;
		bJogFast					:= FALSE;
		fbJogSlowToFastDlyTm.IN		:= FALSE;

		eLifterBtmAct		:= LifterActJogStop;

		IF p_eLifterBtmStat = LifterActJogStop AND p_eLifterBtmStatus = Done THEN
			eLifterBtmAct		:= LifterActIdle;

			bJogStopLifter	:= FALSE;

			tyP1031MagSetTeach.tyMotionStdLifter.tyBtnStop.bRtCompl			:= FALSE;
			tyP1031MagSetTeach.tyMotionStdLifter.tyBtnJogDown.bRtCompl		:= FALSE;
			tyP1031MagSetTeach.tyMotionStdLifter.tyBtnJogUp.bRtCompl		:= FALSE;
			tyP1031MagSetTeach.tyMotionStdLifter.tyBtnOrigin.bRtCompl		:= FALSE;
			tyP1031MagSetTeach.tyMotionStdLifter.tyBtnMovAbs.bRtCompl		:= FALSE;
			tyP1031MagSetTeach.tyMotionStdLifter.tyBtnMovRel.bRtCompl		:= FALSE;

			tyP1031MagSetTeach.tyTeachLifterMag1Slt1Pos.tyBtn2.bRtCompl		:= FALSE;
			tyP1031MagSetTeach.tyTeachLifterMag2Slt1Pos.tyBtn2.bRtCompl		:= FALSE;
			tyP1031MagSetTeach.tyTeachLifterMag3Slt1Pos.tyBtn2.bRtCompl		:= FALSE;

			tyP1031MagSetTeach.tyMotionStdLifter.tyBtnStop.bValue			:= TRUE;
			tyP1031MagSetTeach.tyMotionStdLifter.tyBtnJogDown.bValue		:= FALSE;
			tyP1031MagSetTeach.tyMotionStdLifter.tyBtnJogUp.bValue			:= FALSE;
			tyP1031MagSetTeach.tyMotionStdLifter.tyBtnOrigin.bValue			:= FALSE;
			tyP1031MagSetTeach.tyMotionStdLifter.tyBtnMovAbs.bValue			:= FALSE;
			tyP1031MagSetTeach.tyMotionStdLifter.tyBtnMovRel.bValue			:= FALSE;

			tyP1031MagSetTeach.tyTeachLifterMag1Slt1Pos.tyBtn2.bValue		:= FALSE;
			tyP1031MagSetTeach.tyTeachLifterMag2Slt1Pos.tyBtn2.bValue		:= FALSE;
			tyP1031MagSetTeach.tyTeachLifterMag3Slt1Pos.tyBtn2.bValue		:= FALSE;

			tyP1031MagSetTeach.tyMotionStdLifter.tyBtnStop.bRtLk			:= TRUE;
			tyP1031MagSetTeach.tyMotionStdLifter.tyBtnJogDown.bRtLk			:= FALSE;
			tyP1031MagSetTeach.tyMotionStdLifter.tyBtnJogUp.bRtLk			:= FALSE;
			tyP1031MagSetTeach.tyMotionStdLifter.tyBtnOrigin.bRtLk			:= FALSE;
			tyP1031MagSetTeach.tyMotionStdLifter.tyBtnMovAbs.bRtLk			:= FALSE;
			tyP1031MagSetTeach.tyMotionStdLifter.tyBtnMovRel.bRtLk			:= FALSE;

			tyP1031MagSetTeach.tyTeachLifterMag1Slt1Pos.tyBtn2.bRtLk		:= FALSE;
			tyP1031MagSetTeach.tyTeachLifterMag2Slt1Pos.tyBtn2.bRtLk		:= FALSE;
			tyP1031MagSetTeach.tyTeachLifterMag3Slt1Pos.tyBtn2.bRtLk		:= FALSE;

		END_IF

	ELSIF tyP1031MagSetTeach.tyMotionStdLifter.tyBtnPwr.bRtCompl = TRUE THEN
		tyP1031MagSetTeach.tyMotionStdLifter.tyBtnPwr.bRtLk					:= TRUE;

		IF tyP1031MagSetTeach.tyMotionStdLifter.tyBtnPwr.bValue = TRUE THEN
			eLifterBtmAct		:= LifterActPwrOn;

			IF p_eLifterBtmStat = LifterActPwrOn AND p_eLifterBtmStatus = Done THEN
				eLifterBtmAct	:= LifterActIdle;

				tyP1031MagSetTeach.tyMotionStdLifter.tyBtnPwr.bRtCompl		:= FALSE;
				tyP1031MagSetTeach.tyMotionStdLifter.tyBtnPwr.bRtLk		:= FALSE;
			END_IF
		ELSE
			eLifterBtmAct		:= LifterActPwrOff;

			IF p_eLifterBtmStat = LifterActPwrOff AND p_eLifterBtmStatus = Done THEN
				eLifterBtmAct	:= LifterActIdle;

				tyP1031MagSetTeach.tyMotionStdLifter.tyBtnPwr.bRtCompl		:= FALSE;
				tyP1031MagSetTeach.tyMotionStdLifter.tyBtnPwr.bRtLk		:= FALSE;
			END_IF
		END_IF

	ELSIF tyP1031MagSetTeach.tyMotionStdLifter.tyBtnOrigin.bRtCompl = TRUE THEN
		tyP1031MagSetTeach.tyMotionStdLifter.tyBtnOrigin.bValue				:= TRUE;
		tyP1031MagSetTeach.tyMotionStdLifter.tyBtnStop.bValue					:= FALSE;

		tyP1031MagSetTeach.tyMotionStdLifter.tyBtnOrigin.bRtLk					:= TRUE;
		tyP1031MagSetTeach.tyMotionStdLifter.tyBtnStop.bRtLk					:= FALSE;

		eLifterBtmAct		:= LifterActHoming;

		IF p_eLifterBtmStat = LifterActHoming AND p_eLifterBtmStatus = Done THEN
			eLifterBtmAct	:= LifterActIdle;

			tyP1031MagSetTeach.tyMotionStdLifter.tyBtnOrigin.bRtCompl		:= FALSE;
			tyP1031MagSetTeach.tyMotionStdLifter.tyBtnOrigin.bValue		:= FALSE;
			tyP1031MagSetTeach.tyMotionStdLifter.tyBtnStop.bValue			:= TRUE;

			tyP1031MagSetTeach.tyMotionStdLifter.tyBtnOrigin.bRtLk			:= FALSE;
			tyP1031MagSetTeach.tyMotionStdLifter.tyBtnStop.bRtLk			:= TRUE;

		END_IF

	ELSIF tyP1031MagSetTeach.tyMotionStdLifter.tyBtnRst.bRtCompl = TRUE THEN
		tyP1031MagSetTeach.tyMotionStdLifter.tyBtnRst.bValue				:= TRUE;
		tyP1031MagSetTeach.tyMotionStdLifter.tyBtnRst.bRtLk				:= TRUE;

		eLifterBtmAct		:= LifterActRstAxisErr;

		IF p_eLifterBtmStat = LifterActRstAxisErr AND p_eLifterBtmStatus = Done THEN
			eLifterBtmAct	:= LifterActIdle;

			tyP1031MagSetTeach.tyMotionStdLifter.tyBtnRst.bRtCompl			:= FALSE;
			tyP1031MagSetTeach.tyMotionStdLifter.tyBtnRst.bValue			:= FALSE;
			tyP1031MagSetTeach.tyMotionStdLifter.tyBtnRst.bRtLk			:= FALSE;

			fbLmtRstTm.IN			:= FALSE;
		END_IF

	ELSIF tyP1031MagSetTeach.tyTeachLifterMag1Slt1Pos.tyBtn2.bRtCompl = TRUE THEN
		tyP1031MagSetTeach.tyTeachLifterMag1Slt1Pos.tyBtn2.bValue			:= TRUE;
		tyP1031MagSetTeach.tyMotionStdLifter.tyBtnStop.bValue				:= FALSE;

		tyP1031MagSetTeach.tyTeachLifterMag1Slt1Pos.tyBtn2.bRtLk		:= TRUE;
		tyP1031MagSetTeach.tyMotionStdLifter.tyBtnStop.bRtLk			:= FALSE;

		//diMnlLifterMag1GoSlt	:= 1;
		diMnlLifterMag1GoSlt	:= tyP1031MagSetTeach.tyTeachLifterMag1Slt1Pos.tyNumNewSlt.diValue;
		diMnlLifterNomSpd		:= tyP1031MagSetTeach.tyMotionStdLifter.tyNumNomSpd.diValue;

		eLifterBtmAct		:= LifterActGoASltPos;

		IF p_eLifterBtmStat = LifterActGoASltPos AND p_eLifterBtmStatus = Done THEN
			eLifterBtmAct	:= LifterActIdle;

			tyP1031MagSetTeach.tyTeachLifterMag1Slt1Pos.tyBtn2.bRtCompl			:= FALSE;
			tyP1031MagSetTeach.tyTeachLifterMag1Slt1Pos.tyBtn2.bValue			:= FALSE;
			tyP1031MagSetTeach.tyMotionStdLifter.tyBtnStop.bValue				:= TRUE;

			tyP1031MagSetTeach.tyTeachLifterMag1Slt1Pos.tyBtn2.bRtLk			:= FALSE;
			tyP1031MagSetTeach.tyMotionStdLifter.tyBtnStop.bRtLk				:= TRUE;
		END_IF

	ELSIF tyP1031MagSetTeach.tyTeachLifterMag2Slt1Pos.tyBtn2.bRtCompl = TRUE THEN
		tyP1031MagSetTeach.tyTeachLifterMag2Slt1Pos.tyBtn2.bValue			:= TRUE;
		tyP1031MagSetTeach.tyMotionStdLifter.tyBtnStop.bValue				:= FALSE;

		tyP1031MagSetTeach.tyTeachLifterMag2Slt1Pos.tyBtn2.bRtLk			:= TRUE;
		tyP1031MagSetTeach.tyMotionStdLifter.tyBtnStop.bRtLk				:= FALSE;

		//diMnlLifterMag2GoSlt	:= 1;
		diMnlLifterMag2GoSlt	:= tyP1031MagSetTeach.tyTeachLifterMag2Slt1Pos.tyNumNewSlt.diValue;
		diMnlLifterNomSpd		:= tyP1031MagSetTeach.tyMotionStdLifter.tyNumNomSpd.diValue;

		eLifterBtmAct		:= LifterActGoBSltPos;

		IF p_eLifterBtmStat = LifterActGoBSltPos AND p_eLifterBtmStatus = Done THEN
			eLifterBtmAct	:= LifterActIdle;

			tyP1031MagSetTeach.tyTeachLifterMag2Slt1Pos.tyBtn2.bRtCompl			:= FALSE;
			tyP1031MagSetTeach.tyTeachLifterMag2Slt1Pos.tyBtn2.bValue			:= FALSE;
			tyP1031MagSetTeach.tyMotionStdLifter.tyBtnStop.bValue				:= TRUE;

			tyP1031MagSetTeach.tyTeachLifterMag2Slt1Pos.tyBtn2.bRtLk			:= FALSE;
			tyP1031MagSetTeach.tyMotionStdLifter.tyBtnStop.bRtLk				:= TRUE;
		END_IF

	ELSIF tyP1031MagSetTeach.tyTeachLifterMag3Slt1Pos.tyBtn2.bRtCompl = TRUE THEN
		tyP1031MagSetTeach.tyTeachLifterMag3Slt1Pos.tyBtn2.bValue			:= TRUE;
		tyP1031MagSetTeach.tyMotionStdLifter.tyBtnStop.bValue				:= FALSE;

		tyP1031MagSetTeach.tyTeachLifterMag3Slt1Pos.tyBtn2.bRtLk			:= TRUE;
		tyP1031MagSetTeach.tyMotionStdLifter.tyBtnStop.bRtLk				:= FALSE;

		//diMnlLifterMag3GoSlt	:= 1;
		diMnlLifterMag3GoSlt	:= tyP1031MagSetTeach.tyTeachLifterMag3Slt1Pos.tyNumNewSlt.diValue;
		diMnlLifterNomSpd		:= tyP1031MagSetTeach.tyMotionStdLifter.tyNumNomSpd.diValue;

		eLifterBtmAct		:= LifterActGoCSltPos;

		IF p_eLifterBtmStat = LifterActGoCSltPos AND p_eLifterBtmStatus = Done THEN
			eLifterBtmAct	:= LifterActIdle;

			tyP1031MagSetTeach.tyTeachLifterMag3Slt1Pos.tyBtn2.bRtCompl			:= FALSE;
			tyP1031MagSetTeach.tyTeachLifterMag3Slt1Pos.tyBtn2.bValue			:= FALSE;
			tyP1031MagSetTeach.tyMotionStdLifter.tyBtnStop.bValue				:= TRUE;

			tyP1031MagSetTeach.tyTeachLifterMag3Slt1Pos.tyBtn2.bRtLk			:= FALSE;
			tyP1031MagSetTeach.tyMotionStdLifter.tyBtnStop.bRtLk				:= TRUE;
		END_IF

	ELSIF tyP1031MagSetTeach.tyMotionStdLifter.tyBtnMovAbs.bRtCompl = TRUE THEN

		tyP1031MagSetTeach.tyMotionStdLifter.tyBtnMovAbs.bValue				:= TRUE;
		tyP1031MagSetTeach.tyMotionStdLifter.tyBtnStop.bValue				:= FALSE;

		tyP1031MagSetTeach.tyMotionStdLifter.tyBtnMovAbs.bRtLk				:= TRUE;
		tyP1031MagSetTeach.tyMotionStdLifter.tyBtnStop.bRtLk					:= FALSE;

		diMnlLifterTargetPos	:= tyP1031MagSetTeach.tyMotionStdLifter.tyNumTargetPos.diValue;
		diMnlLifterNomSpd		:= tyP1031MagSetTeach.tyMotionStdLifter.tyNumNomSpd.diValue;

		eLifterBtmAct			:= LifterActMovAbs;

		IF p_eLifterBtmStat = LifterActMovAbs AND p_eLifterBtmStatus = Done THEN
			eLifterBtmAct	:= LifterActIdle;

			tyP1031MagSetTeach.tyMotionStdLifter.tyBtnMovAbs.bRtCompl	:= FALSE;
			tyP1031MagSetTeach.tyMotionStdLifter.tyBtnMovAbs.bValue		:= FALSE;
			tyP1031MagSetTeach.tyMotionStdLifter.tyBtnStop.bValue		:= TRUE;

			tyP1031MagSetTeach.tyMotionStdLifter.tyBtnMovAbs.bRtLk		:= FALSE;
			tyP1031MagSetTeach.tyMotionStdLifter.tyBtnStop.bRtLk		:= TRUE;
		END_IF

	ELSIF tyP1031MagSetTeach.tyMotionStdLifter.tyBtnMovRel.bRtCompl = TRUE THEN
		tyP1031MagSetTeach.tyMotionStdLifter.tyBtnMovRel.bValue			:= TRUE;
		tyP1031MagSetTeach.tyMotionStdLifter.tyBtnStop.bValue			:= FALSE;

		tyP1031MagSetTeach.tyMotionStdLifter.tyBtnMovRel.bRtLk			:= TRUE;
		tyP1031MagSetTeach.tyMotionStdLifter.tyBtnStop.bRtLk				:= FALSE;

		diMnlLifterStepSize		:= tyP1031MagSetTeach.tyMotionStdLifter.tyNumStepSize.diValue;
		diMnlLifterNomSpd		:= tyP1031MagSetTeach.tyMotionStdLifter.tyNumNomSpd.diValue;

		eLifterBtmAct		:= LifterActMovRel;

		IF p_eLifterBtmStat = LifterActMovRel AND p_eLifterBtmStatus = Done THEN
			eLifterBtmAct	:= LifterActIdle;

			tyP1031MagSetTeach.tyMotionStdLifter.tyBtnMovRel.bRtCompl		:= FALSE;
			tyP1031MagSetTeach.tyMotionStdLifter.tyBtnMovRel.bValue			:= FALSE;
			tyP1031MagSetTeach.tyMotionStdLifter.tyBtnStop.bValue			:= TRUE;

			tyP1031MagSetTeach.tyMotionStdLifter.tyBtnMovRel.bRtLk			:= FALSE;
			tyP1031MagSetTeach.tyMotionStdLifter.tyBtnStop.bRtLk				:= TRUE;

		END_IF

	ELSIF (tyP1031MagSetTeach.tyMotionStdLifter.tyBtnJogDown.bValue = TRUE) AND (fbJogSlowToFastDlyTm.Q = FALSE) AND (bJogSlow = FALSE) THEN
		tyP1031MagSetTeach.tyMotionStdLifter.tyBtnStop.bValue				:= FALSE;
		tyP1031MagSetTeach.tyMotionStdLifter.tyBtnStop.bRtLk				:= FALSE;

		fbJogSlowToFastDlyTm.IN		:= TRUE;

		diMnlLifterJogSpd	:= tyP1031MagSetTeach.tyMotionStdLifter.tyNumSlwSpd.diValue;

		eLifterBtmAct		:= LifterActJogDown;

		IF p_eLifterBtmStat = LifterActJogDown AND p_eLifterBtmStatus = Done THEN

			eLifterBtmAct	:= LifterActIdle;
			bJogSlow				:= TRUE;

		ELSIF p_eLifterBtmStatus = Error THEN

			fbJogSlowToFastDlyTm.IN	:= FALSE;
			bJogSlow				:= TRUE;

		END_IF

	ELSIF (tyP1031MagSetTeach.tyMotionStdLifter.tyBtnJogDown.bValue = TRUE) AND (fbJogSlowToFastDlyTm.Q = TRUE) AND (bJogFast = FALSE) THEN
		tyP1031MagSetTeach.tyMotionStdLifter.tyBtnStop.bValue					:= FALSE;
		tyP1031MagSetTeach.tyMotionStdLifter.tyBtnStop.bRtLk					:= FALSE;

		fbJogSlowToFastDlyTm.IN		:= TRUE;

		diMnlLifterJogSpd	:= tyP1031MagSetTeach.tyMotionStdLifter.tyNumNomSpd.diValue;

		eLifterBtmAct		:= LifterActJogDown;

		IF p_eLifterBtmStat = LifterActJogDown AND p_eLifterBtmStatus = Done THEN
			eLifterBtmAct	:= LifterActIdle;
			bJogFast				:= TRUE;
		ELSIF p_eLifterBtmStatus = Error THEN
			fbJogSlowToFastDlyTm.IN	:= FALSE;
			bJogFast				:= TRUE;
		END_IF

	ELSIF (tyP1031MagSetTeach.tyMotionStdLifter.tyBtnJogUp.bValue = TRUE) AND (fbJogSlowToFastDlyTm.Q = FALSE) AND (bJogSlow = FALSE) THEN
		tyP1031MagSetTeach.tyMotionStdLifter.tyBtnStop.bValue				:= FALSE;
		tyP1031MagSetTeach.tyMotionStdLifter.tyBtnStop.bRtLk				:= FALSE;

		fbJogSlowToFastDlyTm.IN		:= TRUE;

		diMnlLifterJogSpd	:= tyP1031MagSetTeach.tyMotionStdLifter.tyNumSlwSpd.diValue;

		eLifterBtmAct		:= LifterActJogUp;

		IF p_eLifterBtmStat = LifterActJogUp AND p_eLifterBtmStatus = Done THEN
			eLifterBtmAct	:= LifterActIdle;
			bJogSlow				:= TRUE;

		ELSIF p_eLifterBtmStatus = Error THEN
			fbJogSlowToFastDlyTm.IN	:= FALSE;
			bJogSlow				:= TRUE;
		END_IF

	ELSIF (tyP1031MagSetTeach.tyMotionStdLifter.tyBtnJogUp.bValue = TRUE) AND (fbJogSlowToFastDlyTm.Q = TRUE) AND (bJogFast = FALSE) THEN

		tyP1031MagSetTeach.tyMotionStdLifter.tyBtnStop.bValue				:= FALSE;
		tyP1031MagSetTeach.tyMotionStdLifter.tyBtnStop.bRtLk					:= FALSE;

		fbJogSlowToFastDlyTm.IN		:= TRUE;

		diMnlLifterJogSpd	:= tyP1031MagSetTeach.tyMotionStdLifter.tyNumNomSpd.diValue;

		eLifterBtmAct		:= LifterActJogUp;

		IF p_eLifterBtmStat = LifterActJogUp AND p_eLifterBtmStatus = Done THEN
			eLifterBtmAct	:= LifterActIdle;
			bJogFast	:= TRUE;

		ELSIF p_eLifterBtmStatus = Error THEN
			fbJogSlowToFastDlyTm.IN	:= FALSE;
			bJogFast				:= TRUE;
		END_IF
	END_IF

	IF tyP1031MagSetTeach.tyInOutletShutterFB.tyBtnOpen.bRtCompl = TRUE THEN
		tyP1031MagSetTeach.tyInOutletShutterFB.tyBtnOpen.bRtCompl	:= FALSE;

		tyP1031MagSetTeach.tyInOutletShutterFB.tyBtnOpen.bValue	:= TRUE;
		tyP1031MagSetTeach.tyInOutletShutterFB.tyBtnClose.bValue	:= FALSE;

	ELSIF tyP1031MagSetTeach.tyInOutletShutterFB.tyBtnClose.bRtCompl = TRUE THEN
		tyP1031MagSetTeach.tyInOutletShutterFB.tyBtnClose.bRtCompl	:= FALSE;

		tyP1031MagSetTeach.tyInOutletShutterFB.tyBtnClose.bValue	:= TRUE;
		tyP1031MagSetTeach.tyInOutletShutterFB.tyBtnOpen.bValue	:= FALSE;
	END_IF

	IF tyP1031MagSetTeach.tyInOutletShutterFB.tyBtnOpen.bValue = TRUE THEN
		eInShutterAct	:= PneuActRet;
		eOutShutterAct	:= PneuActRet;
		eOutShutterAct2	:= PneuActRet;
		eOutShutterAct3	:= PneuActRet;

		IF (p_eInShutterStat = PneuActRet AND p_eInShutterStatus = Done)
			AND (p_eOutShutterStat = PneuActRet AND p_eOutShutterStatus = Done)
			AND (p_eOutShutterStat2 = PneuActRet AND p_eOutShutterStatus2 = Done)
			AND (p_eOutShutterStat3 = PneuActRet AND p_eOutShutterStatus3 = Done)
			THEN
			eInShutterAct	:= PneuActIdle;
			eOutShutterAct	:= PneuActIdle;
			eOutShutterAct2	:= PneuActIdle;
			eOutShutterAct3	:= PneuActIdle;
			tyP1031MagSetTeach.tyInOutletShutterFB.tyBtnOpen.bValue	:= FALSE;
		ELSIF p_eInShutterStatus = Error OR p_eOutShutterStatus = Error OR p_eOutShutterStatus2 = Error OR p_eOutShutterStatus3 = Error THEN
			tyP1031MagSetTeach.tyInOutletShutterFB.tyBtnOpen.bValue	:= FALSE;
		END_IF

	ELSIF tyP1031MagSetTeach.tyInOutletShutterFB.tyBtnClose.bValue = TRUE THEN
		eInShutterAct	:= PneuActExt;
		eOutShutterAct	:= PneuActExt;
		eOutShutterAct2	:= PneuActExt;
		eOutShutterAct3	:= PneuActExt;
		IF (p_eInShutterStat = PneuActExt AND p_eInShutterStatus = Done)
			AND (p_eOutShutterStat = PneuActExt AND p_eOutShutterStatus = Done)
			AND (p_eOutShutterStat2 = PneuActExt AND p_eOutShutterStatus2 = Done)
			AND (p_eOutShutterStat3 = PneuActExt AND p_eOutShutterStatus3 = Done)
			THEN
			eInShutterAct	:= PneuActIdle;
			eOutShutterAct	:= PneuActIdle;
			eOutShutterAct2	:= PneuActIdle;
			eOutShutterAct3	:= PneuActIdle;
			tyP1031MagSetTeach.tyInOutletShutterFB.tyBtnClose.bValue := FALSE;
		ELSIF p_eInShutterStatus = Error OR p_eOutShutterStatus = Error OR p_eOutShutterStatus2 = Error OR p_eOutShutterStatus3 = Error THEN
			tyP1031MagSetTeach.tyInOutletShutterFB.tyBtnClose.bValue := FALSE;
		END_IF
	END_IF

	IF p_eLifterBtmStat = LifterActStop AND (p_eLifterBtmStatus = Done OR p_eLifterBtmStatus = Error) THEN
		eLifterBtmAct	:= LifterActIdle;
	END_IF

	//bypass curtain sensor
	IF bTeachLifterMag1Slt1Pos OR bTeachLifterMag2Slt1Pos OR bTeachLifterMag3Slt1Pos THEN
		bBypCurtainSen			:= tyP1031MagSetTeach.tyTeachLifterMag1Slt1Pos.tyBtn4.bValue OR tyP1031MagSetTeach.tyTeachLifterMag2Slt1Pos.tyBtn4.bValue OR tyP1031MagSetTeach.tyTeachLifterMag3Slt1Pos.tyBtn4.bValue;
		bBypCurtainPBLED		:= tyP1031MagSetTeach.tyTeachLifterMag1Slt1Pos.tyBtn4.bValue OR tyP1031MagSetTeach.tyTeachLifterMag2Slt1Pos.tyBtn4.bValue OR tyP1031MagSetTeach.tyTeachLifterMag3Slt1Pos.tyBtn4.bValue;
	END_IF

END_ACTION
```

#### Act_OptP1031LifterFBStat.st
```iecst
ACTION Act_OptP1031LifterFBStat:

	IF p_bLifterBtmAxisErr = TRUE THEN
		tyP1031MagSetTeach.tyMotionStdLifter.tyStringStat.sValue		:= p_sLifterBtmAxisErrTxt;
	ELSE
		tyP1031MagSetTeach.tyMotionStdLifter.tyStringStat.sValue		:= p_sLifterBtmStatTxt;
	END_IF

END_ACTION
```

#### Act_OptP1031LifterMask.st
```iecst
ACTION Act_OptP1031LifterMask:

	// Interlock Power
	IF p_bLifterBtmAxisErr = TRUE AND p_bLifterBtmPwrOn = FALSE THEN
		fUIInRtStatOff(ADR(tyP1031MagSetTeach.tyMotionStdLifter.tyBtnPwr.uiMaskRtStat));
		tyP1031MagSetTeach.tyMotionStdLifter.tyBtnPwr.bValue		:= FALSE;
	ELSE
		fUIInRtStatHide(ADR(tyP1031MagSetTeach.tyMotionStdLifter.tyBtnPwr.uiMaskRtStat));
	END_IF

	// Interlock Others Move
	IF p_bLifterBtmAxisErr = TRUE OR p_bLifterBtmPwrOn = FALSE THEN
		fUIInRtStatOff(ADR(tyP1031MagSetTeach.tyMotionStdLifter.tyBtnOrigin.uiMaskRtStat));
		fUIInRtStatOff(ADR(tyP1031MagSetTeach.tyMotionStdLifter.tyBtnMovRel.uiMaskRtStat));
		fUIInRtStatOff(ADR(tyP1031MagSetTeach.tyMotionStdLifter.tyBtnJogUp.uiMaskRtStat));
		fUIInRtStatOff(ADR(tyP1031MagSetTeach.tyMotionStdLifter.tyBtnJogDown.uiMaskRtStat));
	ELSE
		fUIInRtStatHide(ADR(tyP1031MagSetTeach.tyMotionStdLifter.tyBtnOrigin.uiMaskRtStat));
		fUIInRtStatHide(ADR(tyP1031MagSetTeach.tyMotionStdLifter.tyBtnMovRel.uiMaskRtStat));
		fUIInRtStatHide(ADR(tyP1031MagSetTeach.tyMotionStdLifter.tyBtnJogUp.uiMaskRtStat));
		fUIInRtStatHide(ADR(tyP1031MagSetTeach.tyMotionStdLifter.tyBtnJogDown.uiMaskRtStat));
	END_IF

	// Interlock Move Absolute
	IF p_bLifterBtmAxisErr = TRUE OR p_bLifterBtmPwrOn = FALSE OR p_bLifterBtmIsHomed = FALSE THEN

		fUIInRtStatOff(ADR(tyP1031MagSetTeach.tyTeachLifterMag1Slt1Pos.tyBtn2.uiMaskRtStat));
		fUIInRtStatOff(ADR(tyP1031MagSetTeach.tyTeachLifterMag2Slt1Pos.tyBtn2.uiMaskRtStat));
		fUIInRtStatOff(ADR(tyP1031MagSetTeach.tyTeachLifterMag3Slt1Pos.tyBtn2.uiMaskRtStat));
		fUIInRtStatOff(ADR(tyP1031MagSetTeach.tyMotionStdLifter.tyBtnMovAbs.uiMaskRtStat));
	ELSE
		fUIInRtStatHide(ADR(tyP1031MagSetTeach.tyTeachLifterMag1Slt1Pos.tyBtn2.uiMaskRtStat));
		fUIInRtStatHide(ADR(tyP1031MagSetTeach.tyTeachLifterMag2Slt1Pos.tyBtn2.uiMaskRtStat));
		fUIInRtStatHide(ADR(tyP1031MagSetTeach.tyTeachLifterMag3Slt1Pos.tyBtn2.uiMaskRtStat));
		fUIInRtStatHide(ADR(tyP1031MagSetTeach.tyMotionStdLifter.tyBtnMovAbs.uiMaskRtStat));
	END_IF

	//Interlock Limit Sensor
	IF tyP1031MagSetTeach.tyMotionStdLifter.tyBtnDownLmtSen.bValue = TRUE THEN
		fUIInRtStatOff(ADR(tyP1031MagSetTeach.tyMotionStdLifter.tyBtnJogDown.uiMaskRtStat));
	END_IF

	IF tyP1031MagSetTeach.tyMotionStdLifter.tyBtnUpLmtSen.bValue = TRUE THEN
		fUIInRtStatOff(ADR(tyP1031MagSetTeach.tyMotionStdLifter.tyBtnJogUp.uiMaskRtStat));
	END_IF

	// Interlock When Moving
	IF tyP1031MagSetTeach.tyMotionStdLifter.tyBtnOrigin.bRtCompl = TRUE THEN
		fUIInRtStatOff(ADR(tyP1031MagSetTeach.tyMotionStdLifter.tyBtnMovAbs.uiMaskRtStat));
		fUIInRtStatOff(ADR(tyP1031MagSetTeach.tyMotionStdLifter.tyBtnMovRel.uiMaskRtStat));
		fUIInRtStatOff(ADR(tyP1031MagSetTeach.tyMotionStdLifter.tyBtnJogUp.uiMaskRtStat));
		fUIInRtStatOff(ADR(tyP1031MagSetTeach.tyMotionStdLifter.tyBtnJogDown.uiMaskRtStat));

		fUIInRtStatOff(ADR(tyP1031MagSetTeach.tyTeachLifterMag1Slt1Pos.tyBtn2.uiMaskRtStat));
		fUIInRtStatOff(ADR(tyP1031MagSetTeach.tyTeachLifterMag2Slt1Pos.tyBtn2.uiMaskRtStat));
		fUIInRtStatOff(ADR(tyP1031MagSetTeach.tyTeachLifterMag3Slt1Pos.tyBtn2.uiMaskRtStat));

	ELSIF tyP1031MagSetTeach.tyMotionStdLifter.tyBtnMovAbs.bRtCompl = TRUE THEN
		fUIInRtStatOff(ADR(tyP1031MagSetTeach.tyMotionStdLifter.tyBtnOrigin.uiMaskRtStat));
		fUIInRtStatOff(ADR(tyP1031MagSetTeach.tyMotionStdLifter.tyBtnMovRel.uiMaskRtStat));
		fUIInRtStatOff(ADR(tyP1031MagSetTeach.tyMotionStdLifter.tyBtnJogUp.uiMaskRtStat));
		fUIInRtStatOff(ADR(tyP1031MagSetTeach.tyMotionStdLifter.tyBtnJogDown.uiMaskRtStat));

		fUIInRtStatOff(ADR(tyP1031MagSetTeach.tyTeachLifterMag1Slt1Pos.tyBtn2.uiMaskRtStat));
		fUIInRtStatOff(ADR(tyP1031MagSetTeach.tyTeachLifterMag2Slt1Pos.tyBtn2.uiMaskRtStat));
		fUIInRtStatOff(ADR(tyP1031MagSetTeach.tyTeachLifterMag3Slt1Pos.tyBtn2.uiMaskRtStat));

	ELSIF tyP1031MagSetTeach.tyMotionStdLifter.tyBtnMovRel.bRtCompl = TRUE THEN
		fUIInRtStatOff(ADR(tyP1031MagSetTeach.tyMotionStdLifter.tyBtnOrigin.uiMaskRtStat));
		fUIInRtStatOff(ADR(tyP1031MagSetTeach.tyMotionStdLifter.tyBtnMovAbs.uiMaskRtStat));
		fUIInRtStatOff(ADR(tyP1031MagSetTeach.tyMotionStdLifter.tyBtnJogUp.uiMaskRtStat));
		fUIInRtStatOff(ADR(tyP1031MagSetTeach.tyMotionStdLifter.tyBtnJogDown.uiMaskRtStat));

		fUIInRtStatOff(ADR(tyP1031MagSetTeach.tyTeachLifterMag1Slt1Pos.tyBtn2.uiMaskRtStat));
		fUIInRtStatOff(ADR(tyP1031MagSetTeach.tyTeachLifterMag2Slt1Pos.tyBtn2.uiMaskRtStat));
		fUIInRtStatOff(ADR(tyP1031MagSetTeach.tyTeachLifterMag3Slt1Pos.tyBtn2.uiMaskRtStat));

	ELSIF tyP1031MagSetTeach.tyMotionStdLifter.tyBtnJogDown.bRtCompl = TRUE OR tyP1031MagSetTeach.tyMotionStdLifter.tyBtnJogDown.bValue = TRUE THEN
		fUIInRtStatOff(ADR(tyP1031MagSetTeach.tyMotionStdLifter.tyBtnOrigin.uiMaskRtStat));
		fUIInRtStatOff(ADR(tyP1031MagSetTeach.tyMotionStdLifter.tyBtnMovAbs.uiMaskRtStat));
		fUIInRtStatOff(ADR(tyP1031MagSetTeach.tyMotionStdLifter.tyBtnMovRel.uiMaskRtStat));
		fUIInRtStatOff(ADR(tyP1031MagSetTeach.tyMotionStdLifter.tyBtnJogUp.uiMaskRtStat));

		fUIInRtStatOff(ADR(tyP1031MagSetTeach.tyTeachLifterMag1Slt1Pos.tyBtn2.uiMaskRtStat));
		fUIInRtStatOff(ADR(tyP1031MagSetTeach.tyTeachLifterMag2Slt1Pos.tyBtn2.uiMaskRtStat));
		fUIInRtStatOff(ADR(tyP1031MagSetTeach.tyTeachLifterMag3Slt1Pos.tyBtn2.uiMaskRtStat));

	ELSIF tyP1031MagSetTeach.tyMotionStdLifter.tyBtnJogUp.bRtCompl = TRUE OR tyP1031MagSetTeach.tyMotionStdLifter.tyBtnJogUp.bValue = TRUE THEN
		fUIInRtStatOff(ADR(tyP1031MagSetTeach.tyMotionStdLifter.tyBtnOrigin.uiMaskRtStat));
		fUIInRtStatOff(ADR(tyP1031MagSetTeach.tyMotionStdLifter.tyBtnMovAbs.uiMaskRtStat));
		fUIInRtStatOff(ADR(tyP1031MagSetTeach.tyMotionStdLifter.tyBtnMovRel.uiMaskRtStat));
		fUIInRtStatOff(ADR(tyP1031MagSetTeach.tyMotionStdLifter.tyBtnJogDown.uiMaskRtStat));

		fUIInRtStatOff(ADR(tyP1031MagSetTeach.tyTeachLifterMag1Slt1Pos.tyBtn2.uiMaskRtStat));
		fUIInRtStatOff(ADR(tyP1031MagSetTeach.tyTeachLifterMag2Slt1Pos.tyBtn2.uiMaskRtStat));
		fUIInRtStatOff(ADR(tyP1031MagSetTeach.tyTeachLifterMag3Slt1Pos.tyBtn2.uiMaskRtStat));

	ELSIF tyP1031MagSetTeach.tyTeachLifterMag1Slt1Pos.tyBtn2.bRtCompl = TRUE THEN
		fUIInRtStatOff(ADR(tyP1031MagSetTeach.tyMotionStdLifter.tyBtnOrigin.uiMaskRtStat));
		fUIInRtStatOff(ADR(tyP1031MagSetTeach.tyMotionStdLifter.tyBtnMovAbs.uiMaskRtStat));
		fUIInRtStatOff(ADR(tyP1031MagSetTeach.tyMotionStdLifter.tyBtnMovRel.uiMaskRtStat));
		fUIInRtStatOff(ADR(tyP1031MagSetTeach.tyMotionStdLifter.tyBtnJogUp.uiMaskRtStat));
		fUIInRtStatOff(ADR(tyP1031MagSetTeach.tyMotionStdLifter.tyBtnJogDown.uiMaskRtStat));

	ELSIF tyP1031MagSetTeach.tyTeachLifterMag2Slt1Pos.tyBtn2.bRtCompl = TRUE THEN
		fUIInRtStatOff(ADR(tyP1031MagSetTeach.tyMotionStdLifter.tyBtnOrigin.uiMaskRtStat));
		fUIInRtStatOff(ADR(tyP1031MagSetTeach.tyMotionStdLifter.tyBtnMovAbs.uiMaskRtStat));
		fUIInRtStatOff(ADR(tyP1031MagSetTeach.tyMotionStdLifter.tyBtnMovRel.uiMaskRtStat));
		fUIInRtStatOff(ADR(tyP1031MagSetTeach.tyMotionStdLifter.tyBtnJogUp.uiMaskRtStat));
		fUIInRtStatOff(ADR(tyP1031MagSetTeach.tyMotionStdLifter.tyBtnJogDown.uiMaskRtStat));

	ELSIF tyP1031MagSetTeach.tyTeachLifterMag3Slt1Pos.tyBtn2.bRtCompl = TRUE THEN
		fUIInRtStatOff(ADR(tyP1031MagSetTeach.tyMotionStdLifter.tyBtnOrigin.uiMaskRtStat));
		fUIInRtStatOff(ADR(tyP1031MagSetTeach.tyMotionStdLifter.tyBtnMovAbs.uiMaskRtStat));
		fUIInRtStatOff(ADR(tyP1031MagSetTeach.tyMotionStdLifter.tyBtnMovRel.uiMaskRtStat));
		fUIInRtStatOff(ADR(tyP1031MagSetTeach.tyMotionStdLifter.tyBtnJogUp.uiMaskRtStat));
		fUIInRtStatOff(ADR(tyP1031MagSetTeach.tyMotionStdLifter.tyBtnJogDown.uiMaskRtStat));

	END_IF

	//Axis Error
	IF tyP1031MagSetTeach.tyMotionStdLifter.tyBtnPwr.bRtCompl = TRUE THEN
		fUIInRtStatOff(ADR(tyP1031MagSetTeach.tyMotionStdLifter.tyBtnRst.uiMaskRtStat));
	ELSE
		fUIInRtStatHide(ADR(tyP1031MagSetTeach.tyMotionStdLifter.tyBtnRst.uiMaskRtStat));
	END_IF

	//Interlock Button Get
	IF p_bLifterBtmAxisErr = TRUE OR p_bLifterBtmIsHomed = FALSE OR p_bLifterBtmFwdLmtSen = TRUE OR p_bLifterBtmRevLmtSen = TRUE THEN
		fUIInRtStatOff(ADR(tyP1031MagSetTeach.tyTeachLifterMag1Slt1Pos.tyBtn1.uiMaskRtStat));
		fUIInRtStatOff(ADR(tyP1031MagSetTeach.tyTeachLifterMag2Slt1Pos.tyBtn1.uiMaskRtStat));
		fUIInRtStatOff(ADR(tyP1031MagSetTeach.tyTeachLifterMag3Slt1Pos.tyBtn1.uiMaskRtStat));
	ELSE
		fUIInRtStatHide(ADR(tyP1031MagSetTeach.tyTeachLifterMag1Slt1Pos.tyBtn1.uiMaskRtStat));
		fUIInRtStatHide(ADR(tyP1031MagSetTeach.tyTeachLifterMag2Slt1Pos.tyBtn1.uiMaskRtStat));
		fUIInRtStatHide(ADR(tyP1031MagSetTeach.tyTeachLifterMag3Slt1Pos.tyBtn1.uiMaskRtStat));
	END_IF

END_ACTION
```

#### Act_OptP1031LifterUpdtDat.st
```iecst
ACTION Act_OptP1031LifterUpdtDat:

	tyP1031MagSetTeach.tyMotionStdLifter.tyNumCurrPos.diValue		:= p_diLifterBtmActualPos;
	tyP1031MagSetTeach.tyMotionStdLifter.tyNumErrCode.diValue		:= UDINT_TO_DINT(p_udiLifterBtmAxisErrID);
	tyP1031MagSetTeach.tyMotionStdLifter.tyBitmapPwr.usiValueIdx	:= BOOL_TO_USINT(p_bLifterBtmPwrOn);
	tyP1031MagSetTeach.tyMotionStdLifter.tyBitmapRst.usiValueIdx	:= BOOL_TO_USINT(NOT p_bLifterBtmAxisErr);
	tyP1031MagSetTeach.tyMotionStdLifter.tyBitmapOrigin.usiValueIdx	:= BOOL_TO_USINT(p_bLifterBtmIsHomed);
	tyP1031MagSetTeach.tyMotionStdLifter.tyBtnUpLmtSen.bValue		:= p_bLifterBtmUpSen;
	tyP1031MagSetTeach.tyMotionStdLifter.tyBtnDownLmtSen.bValue		:= p_bLifterBtmDownSen;

	//Machine Bitmap
	IF p_bLifterBtmIsHomed = TRUE THEN
		IF p_diLifterBtmActualPos <= (p_tyNtParamCurr.tyUILifterTargetPos.diMax / 3) THEN
			tyP1031MagSetTeach.tyMotionStdLifter.tyBitmapMc.uiValueIdx := 2;
		ELSIF p_diLifterBtmActualPos <= (p_tyNtParamCurr.tyUILifterTargetPos.diMax / 3 * 2) THEN
			tyP1031MagSetTeach.tyMotionStdLifter.tyBitmapMc.uiValueIdx := 3;
		ELSE
			tyP1031MagSetTeach.tyMotionStdLifter.tyBitmapMc.uiValueIdx := 4;
		END_IF
	ELSE
		tyP1031MagSetTeach.tyMotionStdLifter.tyBitmapMc.uiValueIdx	:= 2;
	END_IF

	IF p_tyNtParamCurr.eProjMag = ULMagDual THEN
		IF p_tyNtParamCurr.bProjLifterMagPlatform AND p_tyNtParamCurr.bUIConvDirRL THEN
			IF 	tyP1031MagSetTeach.tyMotionStdLifter.tyBitmapMc.uiValueIdx < 700 THEN
				tyP1031MagSetTeach.tyMotionStdLifter.tyBitmapMc.uiValueIdx	:= tyP1031MagSetTeach.tyMotionStdLifter.tyBitmapMc.uiValueIdx + 700;
			END_IF
		ELSIF p_tyNtParamCurr.bProjLifterMagPlatform THEN
			IF p_tyNtParamCurr.bProjMagConvLane1Prep = FALSE THEN
				IF 	tyP1031MagSetTeach.tyMotionStdLifter.tyBitmapMc.uiValueIdx < 600 THEN
					tyP1031MagSetTeach.tyMotionStdLifter.tyBitmapMc.uiValueIdx	:= tyP1031MagSetTeach.tyMotionStdLifter.tyBitmapMc.uiValueIdx + 600;
				END_IF
			ELSE
				IF 	tyP1031MagSetTeach.tyMotionStdLifter.tyBitmapMc.uiValueIdx < 900 THEN
					tyP1031MagSetTeach.tyMotionStdLifter.tyBitmapMc.uiValueIdx	:= tyP1031MagSetTeach.tyMotionStdLifter.tyBitmapMc.uiValueIdx + 900;
				END_IF
			END_IF
		ELSIF p_tyNtParamCurr.bMagAutoVerifyPrep = FALSE THEN
			IF 	tyP1031MagSetTeach.tyMotionStdLifter.tyBitmapMc.uiValueIdx < 100 THEN
				tyP1031MagSetTeach.tyMotionStdLifter.tyBitmapMc.uiValueIdx	:= tyP1031MagSetTeach.tyMotionStdLifter.tyBitmapMc.uiValueIdx + 300;
			END_IF
		ELSE
			IF 	tyP1031MagSetTeach.tyMotionStdLifter.tyBitmapMc.uiValueIdx < 300 THEN
				tyP1031MagSetTeach.tyMotionStdLifter.tyBitmapMc.uiValueIdx	:= tyP1031MagSetTeach.tyMotionStdLifter.tyBitmapMc.uiValueIdx + 300;
			END_IF
		END_IF
	ELSIF p_tyNtParamCurr.eProjMag = ULMagTriple AND p_tyNtParamCurr.bProjLifterMagPlatform THEN
		IF p_tyNtParamCurr.bProjLifterMagPlatform AND p_tyNtParamCurr.bUIConvDirRL THEN
			IF 	tyP1031MagSetTeach.tyMotionStdLifter.tyBitmapMc.uiValueIdx < 800 THEN
				tyP1031MagSetTeach.tyMotionStdLifter.tyBitmapMc.uiValueIdx	:= tyP1031MagSetTeach.tyMotionStdLifter.tyBitmapMc.uiValueIdx + 800;
			END_IF
		ELSIF p_tyNtParamCurr.bProjLifterMagPlatform THEN
			IF 	tyP1031MagSetTeach.tyMotionStdLifter.tyBitmapMc.uiValueIdx < 500 THEN
				tyP1031MagSetTeach.tyMotionStdLifter.tyBitmapMc.uiValueIdx	:= tyP1031MagSetTeach.tyMotionStdLifter.tyBitmapMc.uiValueIdx + 500;
			END_IF
		ELSIF p_tyNtParamCurr.bMagAutoVerifyPrep = TRUE AND p_tyNtParamCurr.bProjMotorizedPusherPrep = FALSE THEN
			IF 	tyP1031MagSetTeach.tyMotionStdLifter.tyBitmapMc.uiValueIdx < 200 THEN
				tyP1031MagSetTeach.tyMotionStdLifter.tyBitmapMc.uiValueIdx	:= tyP1031MagSetTeach.tyMotionStdLifter.tyBitmapMc.uiValueIdx + 200;
			END_IF
		ELSIF p_tyNtParamCurr.bMagAutoVerifyPrep = FALSE AND p_tyNtParamCurr.bProjMotorizedPusherPrep = TRUE THEN
			IF 	tyP1031MagSetTeach.tyMotionStdLifter.tyBitmapMc.uiValueIdx < 400 THEN
				tyP1031MagSetTeach.tyMotionStdLifter.tyBitmapMc.uiValueIdx	:= tyP1031MagSetTeach.tyMotionStdLifter.tyBitmapMc.uiValueIdx + 400;
			END_IF
		END_IF
	END_IF

END_ACTION
```

#### Act_OptP1031Lifter2FBCtrl.st
```iecst
ACTION Act_OptP1031Lifter2FBCtrl:

	fbJogSlowToFastDlyTm.PT	:= T#2s;
	fbJogSlowToFastDlyTm;
	fbLmtRstTm;

	//Lifter Safety Sensor Interruption
	IF EDGENEG(p_tyDI.bLifterSafetyLmtSW1 AND p_tyDI.bLifterSafetyLmtSW2 AND p_tyDI.bLifterTimingBeltSen) THEN
		tyP1031MagSetTeach.tyMotionStdLifter.tyBtnStop.bRtCompl	:= TRUE;
	END_IF

//	IF EDGEPOS((p_udiLifter2AxisErrID = 21570 OR p_udiLifter2AxisErrID = 21571) AND tyP1031MagSetTeach.tyMotionStdLifter.tyBtnJogDown.bValue = FALSE AND tyP1031MagSetTeach.tyMotionStdLifter.tyBtnJogUp.bValue = FALSE) THEN
	IF EDGEPOS((p_bLifter2FwdLmtSen OR p_bLifter2RevLmtSen OR p_udiLifter2AxisErrID = 21570 OR p_udiLifter2AxisErrID = 21571)
		AND tyP1026McSetTeach.tyMotionStdLifter.tyBtnJogDown.bValue = FALSE
		AND tyP1026McSetTeach.tyMotionStdLifter.tyBtnJogUp.bValue = FALSE) THEN
			fbLmtRstTm.IN				:= TRUE;
	END_IF

	IF fbLmtRstTm.Q = TRUE THEN
		tyP1031MagSetTeach.tyMotionStdLifter.tyBtnRst.bRtCompl		:= TRUE;
	END_IF

	IF (tyP1031MagSetTeach.tyMotionStdLifter.tyBtnJogUp.bValue = FALSE AND tyP1031MagSetTeach.tyMotionStdLifter.tyBtnJogDown.bValue = FALSE) AND (p_bLifter2Jogging = TRUE) THEN
		bJogStopLifter	:= TRUE;
	END_IF

	IF tyP1031MagSetTeach.tyMotionStdLifter.tyBtnStop.bRtCompl = TRUE THEN
		eLifter2Act		:= LifterActStop;

		IF p_eLifter2Stat = LifterActStop AND p_eLifter2Status = Done THEN
			eLifter2Act	:= LifterActIdle;

			tyP1031MagSetTeach.tyMotionStdLifter.tyBtnStop.bRtCompl			:= FALSE;
			tyP1031MagSetTeach.tyMotionStdLifter.tyBtnJogDown.bRtCompl		:= FALSE;
			tyP1031MagSetTeach.tyMotionStdLifter.tyBtnJogUp.bRtCompl		:= FALSE;
			tyP1031MagSetTeach.tyMotionStdLifter.tyBtnOrigin.bRtCompl		:= FALSE;
			tyP1031MagSetTeach.tyMotionStdLifter.tyBtnMovAbs.bRtCompl		:= FALSE;
			tyP1031MagSetTeach.tyMotionStdLifter.tyBtnMovRel.bRtCompl		:= FALSE;

			tyP1031MagSetTeach.tyTeachLifterMag1Slt1Pos.tyBtn2.bRtCompl		:= FALSE;
			tyP1031MagSetTeach.tyTeachLifterMag2Slt1Pos.tyBtn2.bRtCompl		:= FALSE;
			tyP1031MagSetTeach.tyTeachLifterMag3Slt1Pos.tyBtn2.bRtCompl		:= FALSE;

			tyP1031MagSetTeach.tyMotionStdLifter.tyBtnStop.bValue			:= TRUE;
			tyP1031MagSetTeach.tyMotionStdLifter.tyBtnJogDown.bValue		:= FALSE;
			tyP1031MagSetTeach.tyMotionStdLifter.tyBtnJogUp.bValue			:= FALSE;
			tyP1031MagSetTeach.tyMotionStdLifter.tyBtnOrigin.bValue			:= FALSE;
			tyP1031MagSetTeach.tyMotionStdLifter.tyBtnMovAbs.bValue			:= FALSE;
			tyP1031MagSetTeach.tyMotionStdLifter.tyBtnMovRel.bValue			:= FALSE;

			tyP1031MagSetTeach.tyTeachLifterMag1Slt1Pos.tyBtn2.bValue		:= FALSE;
			tyP1031MagSetTeach.tyTeachLifterMag2Slt1Pos.tyBtn2.bValue		:= FALSE;
			tyP1031MagSetTeach.tyTeachLifterMag3Slt1Pos.tyBtn2.bValue		:= FALSE;

			tyP1031MagSetTeach.tyMotionStdLifter.tyBtnStop.bRtLk			:= TRUE;
			tyP1031MagSetTeach.tyMotionStdLifter.tyBtnJogDown.bRtLk			:= FALSE;
			tyP1031MagSetTeach.tyMotionStdLifter.tyBtnJogUp.bRtLk			:= FALSE;
			tyP1031MagSetTeach.tyMotionStdLifter.tyBtnOrigin.bRtLk			:= FALSE;
			tyP1031MagSetTeach.tyMotionStdLifter.tyBtnMovAbs.bRtLk			:= FALSE;
			tyP1031MagSetTeach.tyMotionStdLifter.tyBtnMovRel.bRtLk			:= FALSE;

			tyP1031MagSetTeach.tyTeachLifterMag1Slt1Pos.tyBtn2.bRtLk		:= FALSE;
			tyP1031MagSetTeach.tyTeachLifterMag2Slt1Pos.tyBtn2.bRtLk		:= FALSE;
			tyP1031MagSetTeach.tyTeachLifterMag3Slt1Pos.tyBtn2.bRtLk		:= FALSE;

		END_IF

	ELSIF (tyP1031MagSetTeach.tyMotionStdLifter.tyBtnJogDown.bRtCompl = TRUE) OR (tyP1031MagSetTeach.tyMotionStdLifter.tyBtnJogUp.bRtCompl = TRUE) OR (bJogStopLifter = TRUE) THEN
		bJogSlow					:= FALSE;
		bJogFast					:= FALSE;
		fbJogSlowToFastDlyTm.IN		:= FALSE;

		eLifter2Act		:= LifterActJogStop;

		IF p_eLifter2Stat = LifterActJogStop AND p_eLifter2Status = Done THEN
			eLifter2Act		:= LifterActIdle;

			bJogStopLifter	:= FALSE;

			tyP1031MagSetTeach.tyMotionStdLifter.tyBtnStop.bRtCompl			:= FALSE;
			tyP1031MagSetTeach.tyMotionStdLifter.tyBtnJogDown.bRtCompl		:= FALSE;
			tyP1031MagSetTeach.tyMotionStdLifter.tyBtnJogUp.bRtCompl		:= FALSE;
			tyP1031MagSetTeach.tyMotionStdLifter.tyBtnOrigin.bRtCompl		:= FALSE;
			tyP1031MagSetTeach.tyMotionStdLifter.tyBtnMovAbs.bRtCompl		:= FALSE;
			tyP1031MagSetTeach.tyMotionStdLifter.tyBtnMovRel.bRtCompl		:= FALSE;

			tyP1031MagSetTeach.tyTeachLifterMag1Slt1Pos.tyBtn2.bRtCompl		:= FALSE;
			tyP1031MagSetTeach.tyTeachLifterMag2Slt1Pos.tyBtn2.bRtCompl		:= FALSE;
			tyP1031MagSetTeach.tyTeachLifterMag3Slt1Pos.tyBtn2.bRtCompl		:= FALSE;

			tyP1031MagSetTeach.tyMotionStdLifter.tyBtnStop.bValue			:= TRUE;
			tyP1031MagSetTeach.tyMotionStdLifter.tyBtnJogDown.bValue		:= FALSE;
			tyP1031MagSetTeach.tyMotionStdLifter.tyBtnJogUp.bValue			:= FALSE;
			tyP1031MagSetTeach.tyMotionStdLifter.tyBtnOrigin.bValue			:= FALSE;
			tyP1031MagSetTeach.tyMotionStdLifter.tyBtnMovAbs.bValue			:= FALSE;
			tyP1031MagSetTeach.tyMotionStdLifter.tyBtnMovRel.bValue			:= FALSE;

			tyP1031MagSetTeach.tyTeachLifterMag1Slt1Pos.tyBtn2.bValue		:= FALSE;
			tyP1031MagSetTeach.tyTeachLifterMag2Slt1Pos.tyBtn2.bValue		:= FALSE;
			tyP1031MagSetTeach.tyTeachLifterMag3Slt1Pos.tyBtn2.bValue		:= FALSE;

			tyP1031MagSetTeach.tyMotionStdLifter.tyBtnStop.bRtLk			:= TRUE;
			tyP1031MagSetTeach.tyMotionStdLifter.tyBtnJogDown.bRtLk			:= FALSE;
			tyP1031MagSetTeach.tyMotionStdLifter.tyBtnJogUp.bRtLk			:= FALSE;
			tyP1031MagSetTeach.tyMotionStdLifter.tyBtnOrigin.bRtLk			:= FALSE;
			tyP1031MagSetTeach.tyMotionStdLifter.tyBtnMovAbs.bRtLk			:= FALSE;
			tyP1031MagSetTeach.tyMotionStdLifter.tyBtnMovRel.bRtLk			:= FALSE;

			tyP1031MagSetTeach.tyTeachLifterMag1Slt1Pos.tyBtn2.bRtLk		:= FALSE;
			tyP1031MagSetTeach.tyTeachLifterMag2Slt1Pos.tyBtn2.bRtLk		:= FALSE;
			tyP1031MagSetTeach.tyTeachLifterMag3Slt1Pos.tyBtn2.bRtLk		:= FALSE;

		END_IF

	ELSIF tyP1031MagSetTeach.tyMotionStdLifter.tyBtnPwr.bRtCompl = TRUE THEN
		tyP1031MagSetTeach.tyMotionStdLifter.tyBtnPwr.bRtLk					:= TRUE;

		IF tyP1031MagSetTeach.tyMotionStdLifter.tyBtnPwr.bValue = TRUE THEN
			eLifter2Act		:= LifterActPwrOn;

			IF p_eLifter2Stat = LifterActPwrOn AND p_eLifter2Status = Done THEN
				eLifter2Act	:= LifterActIdle;

				tyP1031MagSetTeach.tyMotionStdLifter.tyBtnPwr.bRtCompl		:= FALSE;
				tyP1031MagSetTeach.tyMotionStdLifter.tyBtnPwr.bRtLk		:= FALSE;
			END_IF
		ELSE
			eLifter2Act		:= LifterActPwrOff;

			IF p_eLifter2Stat = LifterActPwrOff AND p_eLifter2Status = Done THEN
				eLifter2Act	:= LifterActIdle;

				tyP1031MagSetTeach.tyMotionStdLifter.tyBtnPwr.bRtCompl		:= FALSE;
				tyP1031MagSetTeach.tyMotionStdLifter.tyBtnPwr.bRtLk		:= FALSE;
			END_IF
		END_IF

	ELSIF tyP1031MagSetTeach.tyMotionStdLifter.tyBtnOrigin.bRtCompl = TRUE THEN
		tyP1031MagSetTeach.tyMotionStdLifter.tyBtnOrigin.bValue				:= TRUE;
		tyP1031MagSetTeach.tyMotionStdLifter.tyBtnStop.bValue					:= FALSE;

		tyP1031MagSetTeach.tyMotionStdLifter.tyBtnOrigin.bRtLk					:= TRUE;
		tyP1031MagSetTeach.tyMotionStdLifter.tyBtnStop.bRtLk					:= FALSE;

		eLifter2Act		:= LifterActHoming;

		IF p_eLifter2Stat = LifterActHoming AND p_eLifter2Status = Done THEN
			eLifter2Act	:= LifterActIdle;

			tyP1031MagSetTeach.tyMotionStdLifter.tyBtnOrigin.bRtCompl		:= FALSE;
			tyP1031MagSetTeach.tyMotionStdLifter.tyBtnOrigin.bValue		:= FALSE;
			tyP1031MagSetTeach.tyMotionStdLifter.tyBtnStop.bValue			:= TRUE;

			tyP1031MagSetTeach.tyMotionStdLifter.tyBtnOrigin.bRtLk			:= FALSE;
			tyP1031MagSetTeach.tyMotionStdLifter.tyBtnStop.bRtLk			:= TRUE;

		END_IF

	ELSIF tyP1031MagSetTeach.tyMotionStdLifter.tyBtnRst.bRtCompl = TRUE THEN
		tyP1031MagSetTeach.tyMotionStdLifter.tyBtnRst.bValue				:= TRUE;
		tyP1031MagSetTeach.tyMotionStdLifter.tyBtnRst.bRtLk				:= TRUE;

		eLifter2Act		:= LifterActRstAxisErr;

		IF p_eLifter2Stat = LifterActRstAxisErr AND p_eLifter2Status = Done THEN
			eLifter2Act	:= LifterActIdle;

			tyP1031MagSetTeach.tyMotionStdLifter.tyBtnRst.bRtCompl			:= FALSE;
			tyP1031MagSetTeach.tyMotionStdLifter.tyBtnRst.bValue			:= FALSE;
			tyP1031MagSetTeach.tyMotionStdLifter.tyBtnRst.bRtLk			:= FALSE;

			fbLmtRstTm.IN			:= FALSE;
		END_IF

	ELSIF tyP1031MagSetTeach.tyTeachLifterMag1Slt1Pos.tyBtn2.bRtCompl = TRUE THEN
		tyP1031MagSetTeach.tyTeachLifterMag1Slt1Pos.tyBtn2.bValue			:= TRUE;
		tyP1031MagSetTeach.tyMotionStdLifter.tyBtnStop.bValue				:= FALSE;

		tyP1031MagSetTeach.tyTeachLifterMag1Slt1Pos.tyBtn2.bRtLk		:= TRUE;
		tyP1031MagSetTeach.tyMotionStdLifter.tyBtnStop.bRtLk			:= FALSE;

		//diMnlLifterMag1GoSlt	:= 1;
		diMnlLifterMag1GoSlt2	:= tyP1031MagSetTeach.tyTeachLifterMag1Slt1Pos.tyNumNewSlt.diValue;
		diMnlLifterNomSpd2		:= tyP1031MagSetTeach.tyMotionStdLifter.tyNumNomSpd.diValue;

		eLifter2Act		:= LifterActGoASltPos;

		IF p_eLifter2Stat = LifterActGoASltPos AND p_eLifter2Status = Done THEN
			eLifter2Act	:= LifterActIdle;

			tyP1031MagSetTeach.tyTeachLifterMag1Slt1Pos.tyBtn2.bRtCompl			:= FALSE;
			tyP1031MagSetTeach.tyTeachLifterMag1Slt1Pos.tyBtn2.bValue			:= FALSE;
			tyP1031MagSetTeach.tyMotionStdLifter.tyBtnStop.bValue				:= TRUE;

			tyP1031MagSetTeach.tyTeachLifterMag1Slt1Pos.tyBtn2.bRtLk			:= FALSE;
			tyP1031MagSetTeach.tyMotionStdLifter.tyBtnStop.bRtLk				:= TRUE;
		END_IF

	ELSIF tyP1031MagSetTeach.tyTeachLifterMag2Slt1Pos.tyBtn2.bRtCompl = TRUE THEN
		tyP1031MagSetTeach.tyTeachLifterMag2Slt1Pos.tyBtn2.bValue			:= TRUE;
		tyP1031MagSetTeach.tyMotionStdLifter.tyBtnStop.bValue				:= FALSE;

		tyP1031MagSetTeach.tyTeachLifterMag2Slt1Pos.tyBtn2.bRtLk			:= TRUE;
		tyP1031MagSetTeach.tyMotionStdLifter.tyBtnStop.bRtLk				:= FALSE;

		//diMnlLifterMag2GoSlt	:= 1;
		diMnlLifterMag2GoSlt2	:= tyP1031MagSetTeach.tyTeachLifterMag2Slt1Pos.tyNumNewSlt.diValue;
		diMnlLifterNomSpd2		:= tyP1031MagSetTeach.tyMotionStdLifter.tyNumNomSpd.diValue;

		eLifter2Act		:= LifterActGoBSltPos;

		IF p_eLifter2Stat = LifterActGoBSltPos AND p_eLifter2Status = Done THEN
			eLifter2Act	:= LifterActIdle;

			tyP1031MagSetTeach.tyTeachLifterMag2Slt1Pos.tyBtn2.bRtCompl			:= FALSE;
			tyP1031MagSetTeach.tyTeachLifterMag2Slt1Pos.tyBtn2.bValue			:= FALSE;
			tyP1031MagSetTeach.tyMotionStdLifter.tyBtnStop.bValue				:= TRUE;

			tyP1031MagSetTeach.tyTeachLifterMag2Slt1Pos.tyBtn2.bRtLk			:= FALSE;
			tyP1031MagSetTeach.tyMotionStdLifter.tyBtnStop.bRtLk				:= TRUE;
		END_IF

	ELSIF tyP1031MagSetTeach.tyTeachLifterMag3Slt1Pos.tyBtn2.bRtCompl = TRUE THEN
		tyP1031MagSetTeach.tyTeachLifterMag3Slt1Pos.tyBtn2.bValue			:= TRUE;
		tyP1031MagSetTeach.tyMotionStdLifter.tyBtnStop.bValue				:= FALSE;

		tyP1031MagSetTeach.tyTeachLifterMag3Slt1Pos.tyBtn2.bRtLk			:= TRUE;
		tyP1031MagSetTeach.tyMotionStdLifter.tyBtnStop.bRtLk				:= FALSE;

		//diMnlLifterMag3GoSlt	:= 1;
		diMnlLifterMag3GoSlt2	:= tyP1031MagSetTeach.tyTeachLifterMag3Slt1Pos.tyNumNewSlt.diValue;
		diMnlLifterNomSpd2		:= tyP1031MagSetTeach.tyMotionStdLifter.tyNumNomSpd.diValue;

		eLifter2Act		:= LifterActGoCSltPos;

		IF p_eLifter2Stat = LifterActGoCSltPos AND p_eLifter2Status = Done THEN
			eLifter2Act	:= LifterActIdle;

			tyP1031MagSetTeach.tyTeachLifterMag3Slt1Pos.tyBtn2.bRtCompl			:= FALSE;
			tyP1031MagSetTeach.tyTeachLifterMag3Slt1Pos.tyBtn2.bValue			:= FALSE;
			tyP1031MagSetTeach.tyMotionStdLifter.tyBtnStop.bValue				:= TRUE;

			tyP1031MagSetTeach.tyTeachLifterMag3Slt1Pos.tyBtn2.bRtLk			:= FALSE;
			tyP1031MagSetTeach.tyMotionStdLifter.tyBtnStop.bRtLk				:= TRUE;
		END_IF

	ELSIF tyP1031MagSetTeach.tyMotionStdLifter.tyBtnMovAbs.bRtCompl = TRUE THEN

		tyP1031MagSetTeach.tyMotionStdLifter.tyBtnMovAbs.bValue				:= TRUE;
		tyP1031MagSetTeach.tyMotionStdLifter.tyBtnStop.bValue				:= FALSE;

		tyP1031MagSetTeach.tyMotionStdLifter.tyBtnMovAbs.bRtLk				:= TRUE;
		tyP1031MagSetTeach.tyMotionStdLifter.tyBtnStop.bRtLk					:= FALSE;

		diMnlLifterTargetPos2	:= tyP1031MagSetTeach.tyMotionStdLifter.tyNumTargetPos.diValue;
		diMnlLifterNomSpd2		:= tyP1031MagSetTeach.tyMotionStdLifter.tyNumNomSpd.diValue;

		eLifter2Act			:= LifterActMovAbs;

		IF p_eLifter2Stat = LifterActMovAbs AND p_eLifter2Status = Done THEN
			eLifter2Act	:= LifterActIdle;

			tyP1031MagSetTeach.tyMotionStdLifter.tyBtnMovAbs.bRtCompl	:= FALSE;
			tyP1031MagSetTeach.tyMotionStdLifter.tyBtnMovAbs.bValue		:= FALSE;
			tyP1031MagSetTeach.tyMotionStdLifter.tyBtnStop.bValue		:= TRUE;

			tyP1031MagSetTeach.tyMotionStdLifter.tyBtnMovAbs.bRtLk		:= FALSE;
			tyP1031MagSetTeach.tyMotionStdLifter.tyBtnStop.bRtLk		:= TRUE;
		END_IF

	ELSIF tyP1031MagSetTeach.tyMotionStdLifter.tyBtnMovRel.bRtCompl = TRUE THEN
		tyP1031MagSetTeach.tyMotionStdLifter.tyBtnMovRel.bValue			:= TRUE;
		tyP1031MagSetTeach.tyMotionStdLifter.tyBtnStop.bValue			:= FALSE;

		tyP1031MagSetTeach.tyMotionStdLifter.tyBtnMovRel.bRtLk			:= TRUE;
		tyP1031MagSetTeach.tyMotionStdLifter.tyBtnStop.bRtLk				:= FALSE;

		diMnlLifterStepSize2		:= tyP1031MagSetTeach.tyMotionStdLifter.tyNumStepSize.diValue;
		diMnlLifterNomSpd2		:= tyP1031MagSetTeach.tyMotionStdLifter.tyNumNomSpd.diValue;

		eLifter2Act		:= LifterActMovRel;

		IF p_eLifter2Stat = LifterActMovRel AND p_eLifter2Status = Done THEN
			eLifter2Act	:= LifterActIdle;

			tyP1031MagSetTeach.tyMotionStdLifter.tyBtnMovRel.bRtCompl		:= FALSE;
			tyP1031MagSetTeach.tyMotionStdLifter.tyBtnMovRel.bValue			:= FALSE;
			tyP1031MagSetTeach.tyMotionStdLifter.tyBtnStop.bValue			:= TRUE;

			tyP1031MagSetTeach.tyMotionStdLifter.tyBtnMovRel.bRtLk			:= FALSE;
			tyP1031MagSetTeach.tyMotionStdLifter.tyBtnStop.bRtLk				:= TRUE;

		END_IF

	ELSIF (tyP1031MagSetTeach.tyMotionStdLifter.tyBtnJogDown.bValue = TRUE) AND (fbJogSlowToFastDlyTm.Q = FALSE) AND (bJogSlow = FALSE) THEN
		tyP1031MagSetTeach.tyMotionStdLifter.tyBtnStop.bValue				:= FALSE;
		tyP1031MagSetTeach.tyMotionStdLifter.tyBtnStop.bRtLk				:= FALSE;

		fbJogSlowToFastDlyTm.IN		:= TRUE;

		diMnlLifterJogSpd2	:= tyP1031MagSetTeach.tyMotionStdLifter.tyNumSlwSpd.diValue;

		eLifter2Act		:= LifterActJogDown;

		IF p_eLifter2Stat = LifterActJogDown AND p_eLifter2Status = Done THEN

			eLifter2Act	:= LifterActIdle;
			bJogSlow				:= TRUE;

		ELSIF p_eLifter2Status = Error THEN

			fbJogSlowToFastDlyTm.IN	:= FALSE;
			bJogSlow				:= TRUE;

		END_IF

	ELSIF (tyP1031MagSetTeach.tyMotionStdLifter.tyBtnJogDown.bValue = TRUE) AND (fbJogSlowToFastDlyTm.Q = TRUE) AND (bJogFast = FALSE) THEN
		tyP1031MagSetTeach.tyMotionStdLifter.tyBtnStop.bValue					:= FALSE;
		tyP1031MagSetTeach.tyMotionStdLifter.tyBtnStop.bRtLk					:= FALSE;

		fbJogSlowToFastDlyTm.IN		:= TRUE;

		diMnlLifterJogSpd2	:= tyP1031MagSetTeach.tyMotionStdLifter.tyNumNomSpd.diValue;

		eLifter2Act		:= LifterActJogDown;

		IF p_eLifter2Stat = LifterActJogDown AND p_eLifter2Status = Done THEN
			eLifter2Act	:= LifterActIdle;
			bJogFast				:= TRUE;
		ELSIF p_eLifter2Status = Error THEN
			fbJogSlowToFastDlyTm.IN	:= FALSE;
			bJogFast				:= TRUE;
		END_IF

	ELSIF (tyP1031MagSetTeach.tyMotionStdLifter.tyBtnJogUp.bValue = TRUE) AND (fbJogSlowToFastDlyTm.Q = FALSE) AND (bJogSlow = FALSE) THEN
		tyP1031MagSetTeach.tyMotionStdLifter.tyBtnStop.bValue				:= FALSE;
		tyP1031MagSetTeach.tyMotionStdLifter.tyBtnStop.bRtLk				:= FALSE;

		fbJogSlowToFastDlyTm.IN		:= TRUE;

		diMnlLifterJogSpd2	:= tyP1031MagSetTeach.tyMotionStdLifter.tyNumSlwSpd.diValue;

		eLifter2Act		:= LifterActJogUp;

		IF p_eLifter2Stat = LifterActJogUp AND p_eLifter2Status = Done THEN
			eLifter2Act	:= LifterActIdle;
			bJogSlow				:= TRUE;

		ELSIF p_eLifter2Status = Error THEN
			fbJogSlowToFastDlyTm.IN	:= FALSE;
			bJogSlow				:= TRUE;
		END_IF

	ELSIF (tyP1031MagSetTeach.tyMotionStdLifter.tyBtnJogUp.bValue = TRUE) AND (fbJogSlowToFastDlyTm.Q = TRUE) AND (bJogFast = FALSE) THEN

		tyP1031MagSetTeach.tyMotionStdLifter.tyBtnStop.bValue				:= FALSE;
		tyP1031MagSetTeach.tyMotionStdLifter.tyBtnStop.bRtLk					:= FALSE;

		fbJogSlowToFastDlyTm.IN		:= TRUE;

		diMnlLifterJogSpd2	:= tyP1031MagSetTeach.tyMotionStdLifter.tyNumNomSpd.diValue;

		eLifter2Act		:= LifterActJogUp;

		IF p_eLifter2Stat = LifterActJogUp AND p_eLifter2Status = Done THEN
			eLifter2Act	:= LifterActIdle;
			bJogFast	:= TRUE;

		ELSIF p_eLifter2Status = Error THEN
			fbJogSlowToFastDlyTm.IN	:= FALSE;
			bJogFast				:= TRUE;
		END_IF
	END_IF

	IF tyP1031MagSetTeach.tyInOutletShutterFB.tyBtnOpen.bRtCompl = TRUE THEN
		tyP1031MagSetTeach.tyInOutletShutterFB.tyBtnOpen.bRtCompl	:= FALSE;

		tyP1031MagSetTeach.tyInOutletShutterFB.tyBtnOpen.bValue	:= TRUE;
		tyP1031MagSetTeach.tyInOutletShutterFB.tyBtnClose.bValue	:= FALSE;

	ELSIF tyP1031MagSetTeach.tyInOutletShutterFB.tyBtnClose.bRtCompl = TRUE THEN
		tyP1031MagSetTeach.tyInOutletShutterFB.tyBtnClose.bRtCompl	:= FALSE;

		tyP1031MagSetTeach.tyInOutletShutterFB.tyBtnClose.bValue	:= TRUE;
		tyP1031MagSetTeach.tyInOutletShutterFB.tyBtnOpen.bValue	:= FALSE;
	END_IF

	IF tyP1031MagSetTeach.tyInOutletShutterFB.tyBtnOpen.bValue = TRUE THEN
		eInShutterAct	:= PneuActRet;
		eOutShutterAct	:= PneuActRet;
		eOutShutterAct2	:= PneuActRet;
		eOutShutterAct3	:= PneuActRet;

		IF (p_eInShutterStat = PneuActRet AND p_eInShutterStatus = Done)
			AND (p_eOutShutterStat = PneuActRet AND p_eOutShutterStatus = Done)
			AND (p_eOutShutterStat2 = PneuActRet AND p_eOutShutterStatus2 = Done)
			AND (p_eOutShutterStat3 = PneuActRet AND p_eOutShutterStatus3 = Done)
			THEN
			eInShutterAct	:= PneuActIdle;
			eOutShutterAct	:= PneuActIdle;
			eOutShutterAct2	:= PneuActIdle;
			eOutShutterAct3	:= PneuActIdle;
			tyP1031MagSetTeach.tyInOutletShutterFB.tyBtnOpen.bValue	:= FALSE;
		ELSIF p_eInShutterStatus = Error OR p_eOutShutterStatus = Error OR p_eOutShutterStatus2 = Error OR p_eOutShutterStatus3 = Error THEN
			tyP1031MagSetTeach.tyInOutletShutterFB.tyBtnOpen.bValue	:= FALSE;
		END_IF

	ELSIF tyP1031MagSetTeach.tyInOutletShutterFB.tyBtnClose.bValue = TRUE THEN
		eInShutterAct	:= PneuActExt;
		eOutShutterAct	:= PneuActExt;
		eOutShutterAct2	:= PneuActExt;
		eOutShutterAct3	:= PneuActExt;
		IF (p_eInShutterStat = PneuActExt AND p_eInShutterStatus = Done)
			AND (p_eOutShutterStat = PneuActExt AND p_eOutShutterStatus = Done)
			AND (p_eOutShutterStat2 = PneuActExt AND p_eOutShutterStatus2 = Done)
			AND (p_eOutShutterStat3 = PneuActExt AND p_eOutShutterStatus3 = Done)
			THEN
			eInShutterAct	:= PneuActIdle;
			eOutShutterAct	:= PneuActIdle;
			eOutShutterAct2	:= PneuActIdle;
			eOutShutterAct3	:= PneuActIdle;
			tyP1031MagSetTeach.tyInOutletShutterFB.tyBtnClose.bValue := FALSE;
		ELSIF p_eInShutterStatus = Error OR p_eOutShutterStatus = Error OR p_eOutShutterStatus2 = Error OR p_eOutShutterStatus3 = Error THEN
			tyP1031MagSetTeach.tyInOutletShutterFB.tyBtnClose.bValue := FALSE;
		END_IF
	END_IF

	IF p_eLifter2Stat = LifterActStop AND (p_eLifter2Status = Done OR p_eLifter2Status = Error) THEN
		eLifter2Act	:= LifterActIdle;
	END_IF

END_ACTION
```

#### Act_OptP1031Lifter2FBStat.st
```iecst
ACTION Act_OptP1031Lifter2FBStat:

	IF p_bLifter2AxisErr = TRUE THEN
		tyP1031MagSetTeach.tyMotionStdLifter.tyStringStat.sValue		:= p_sLifter2AxisErrTxt;
	ELSE
		tyP1031MagSetTeach.tyMotionStdLifter.tyStringStat.sValue		:= p_sLifter2StatTxt;
	END_IF

END_ACTION
```

#### Act_OptP1031Lifter2Mask.st
```iecst
ACTION Act_OptP1031Lifter2Mask:

	// Interlock Power
	IF p_bLifter2AxisErr = TRUE AND p_bLifter2PwrOn = FALSE THEN
		fUIInRtStatOff(ADR(tyP1031MagSetTeach.tyMotionStdLifter.tyBtnPwr.uiMaskRtStat));
		tyP1031MagSetTeach.tyMotionStdLifter.tyBtnPwr.bValue		:= FALSE;
	ELSE
		fUIInRtStatHide(ADR(tyP1031MagSetTeach.tyMotionStdLifter.tyBtnPwr.uiMaskRtStat));
	END_IF

	// Interlock Others Move
	IF p_bLifter2AxisErr = TRUE OR p_bLifter2PwrOn = FALSE THEN
		fUIInRtStatOff(ADR(tyP1031MagSetTeach.tyMotionStdLifter.tyBtnOrigin.uiMaskRtStat));
		fUIInRtStatOff(ADR(tyP1031MagSetTeach.tyMotionStdLifter.tyBtnMovRel.uiMaskRtStat));
		fUIInRtStatOff(ADR(tyP1031MagSetTeach.tyMotionStdLifter.tyBtnJogUp.uiMaskRtStat));
		fUIInRtStatOff(ADR(tyP1031MagSetTeach.tyMotionStdLifter.tyBtnJogDown.uiMaskRtStat));
	ELSE
		fUIInRtStatHide(ADR(tyP1031MagSetTeach.tyMotionStdLifter.tyBtnOrigin.uiMaskRtStat));
		fUIInRtStatHide(ADR(tyP1031MagSetTeach.tyMotionStdLifter.tyBtnMovRel.uiMaskRtStat));
		fUIInRtStatHide(ADR(tyP1031MagSetTeach.tyMotionStdLifter.tyBtnJogUp.uiMaskRtStat));
		fUIInRtStatHide(ADR(tyP1031MagSetTeach.tyMotionStdLifter.tyBtnJogDown.uiMaskRtStat));
	END_IF

	// Interlock Move Absolute
	IF p_bLifter2AxisErr = TRUE OR p_bLifter2PwrOn = FALSE OR p_bLifter2IsHomed = FALSE THEN

		fUIInRtStatOff(ADR(tyP1031MagSetTeach.tyTeachLifterMag1Slt1Pos.tyBtn2.uiMaskRtStat));
		fUIInRtStatOff(ADR(tyP1031MagSetTeach.tyTeachLifterMag2Slt1Pos.tyBtn2.uiMaskRtStat));
		fUIInRtStatOff(ADR(tyP1031MagSetTeach.tyTeachLifterMag3Slt1Pos.tyBtn2.uiMaskRtStat));
		fUIInRtStatOff(ADR(tyP1031MagSetTeach.tyMotionStdLifter.tyBtnMovAbs.uiMaskRtStat));
	ELSE
		fUIInRtStatHide(ADR(tyP1031MagSetTeach.tyTeachLifterMag1Slt1Pos.tyBtn2.uiMaskRtStat));
		fUIInRtStatHide(ADR(tyP1031MagSetTeach.tyTeachLifterMag2Slt1Pos.tyBtn2.uiMaskRtStat));
		fUIInRtStatHide(ADR(tyP1031MagSetTeach.tyTeachLifterMag3Slt1Pos.tyBtn2.uiMaskRtStat));
		fUIInRtStatHide(ADR(tyP1031MagSetTeach.tyMotionStdLifter.tyBtnMovAbs.uiMaskRtStat));
	END_IF

	//Interlock Limit Sensor
	IF tyP1031MagSetTeach.tyMotionStdLifter.tyBtnDownLmtSen.bValue = TRUE THEN
		fUIInRtStatOff(ADR(tyP1031MagSetTeach.tyMotionStdLifter.tyBtnJogDown.uiMaskRtStat));
	END_IF

	IF tyP1031MagSetTeach.tyMotionStdLifter.tyBtnUpLmtSen.bValue = TRUE THEN
		fUIInRtStatOff(ADR(tyP1031MagSetTeach.tyMotionStdLifter.tyBtnJogUp.uiMaskRtStat));
	END_IF

	// Interlock When Moving
	IF tyP1031MagSetTeach.tyMotionStdLifter.tyBtnOrigin.bRtCompl = TRUE THEN
		fUIInRtStatOff(ADR(tyP1031MagSetTeach.tyMotionStdLifter.tyBtnMovAbs.uiMaskRtStat));
		fUIInRtStatOff(ADR(tyP1031MagSetTeach.tyMotionStdLifter.tyBtnMovRel.uiMaskRtStat));
		fUIInRtStatOff(ADR(tyP1031MagSetTeach.tyMotionStdLifter.tyBtnJogUp.uiMaskRtStat));
		fUIInRtStatOff(ADR(tyP1031MagSetTeach.tyMotionStdLifter.tyBtnJogDown.uiMaskRtStat));

		fUIInRtStatOff(ADR(tyP1031MagSetTeach.tyTeachLifterMag1Slt1Pos.tyBtn2.uiMaskRtStat));
		fUIInRtStatOff(ADR(tyP1031MagSetTeach.tyTeachLifterMag2Slt1Pos.tyBtn2.uiMaskRtStat));
		fUIInRtStatOff(ADR(tyP1031MagSetTeach.tyTeachLifterMag3Slt1Pos.tyBtn2.uiMaskRtStat));

	ELSIF tyP1031MagSetTeach.tyMotionStdLifter.tyBtnMovAbs.bRtCompl = TRUE THEN
		fUIInRtStatOff(ADR(tyP1031MagSetTeach.tyMotionStdLifter.tyBtnOrigin.uiMaskRtStat));
		fUIInRtStatOff(ADR(tyP1031MagSetTeach.tyMotionStdLifter.tyBtnMovRel.uiMaskRtStat));
		fUIInRtStatOff(ADR(tyP1031MagSetTeach.tyMotionStdLifter.tyBtnJogUp.uiMaskRtStat));
		fUIInRtStatOff(ADR(tyP1031MagSetTeach.tyMotionStdLifter.tyBtnJogDown.uiMaskRtStat));

		fUIInRtStatOff(ADR(tyP1031MagSetTeach.tyTeachLifterMag1Slt1Pos.tyBtn2.uiMaskRtStat));
		fUIInRtStatOff(ADR(tyP1031MagSetTeach.tyTeachLifterMag2Slt1Pos.tyBtn2.uiMaskRtStat));
		fUIInRtStatOff(ADR(tyP1031MagSetTeach.tyTeachLifterMag3Slt1Pos.tyBtn2.uiMaskRtStat));

	ELSIF tyP1031MagSetTeach.tyMotionStdLifter.tyBtnMovRel.bRtCompl = TRUE THEN
		fUIInRtStatOff(ADR(tyP1031MagSetTeach.tyMotionStdLifter.tyBtnOrigin.uiMaskRtStat));
		fUIInRtStatOff(ADR(tyP1031MagSetTeach.tyMotionStdLifter.tyBtnMovAbs.uiMaskRtStat));
		fUIInRtStatOff(ADR(tyP1031MagSetTeach.tyMotionStdLifter.tyBtnJogUp.uiMaskRtStat));
		fUIInRtStatOff(ADR(tyP1031MagSetTeach.tyMotionStdLifter.tyBtnJogDown.uiMaskRtStat));

		fUIInRtStatOff(ADR(tyP1031MagSetTeach.tyTeachLifterMag1Slt1Pos.tyBtn2.uiMaskRtStat));
		fUIInRtStatOff(ADR(tyP1031MagSetTeach.tyTeachLifterMag2Slt1Pos.tyBtn2.uiMaskRtStat));
		fUIInRtStatOff(ADR(tyP1031MagSetTeach.tyTeachLifterMag3Slt1Pos.tyBtn2.uiMaskRtStat));

	ELSIF tyP1031MagSetTeach.tyMotionStdLifter.tyBtnJogDown.bRtCompl = TRUE OR tyP1031MagSetTeach.tyMotionStdLifter.tyBtnJogDown.bValue = TRUE THEN
		fUIInRtStatOff(ADR(tyP1031MagSetTeach.tyMotionStdLifter.tyBtnOrigin.uiMaskRtStat));
		fUIInRtStatOff(ADR(tyP1031MagSetTeach.tyMotionStdLifter.tyBtnMovAbs.uiMaskRtStat));
		fUIInRtStatOff(ADR(tyP1031MagSetTeach.tyMotionStdLifter.tyBtnMovRel.uiMaskRtStat));
		fUIInRtStatOff(ADR(tyP1031MagSetTeach.tyMotionStdLifter.tyBtnJogUp.uiMaskRtStat));

		fUIInRtStatOff(ADR(tyP1031MagSetTeach.tyTeachLifterMag1Slt1Pos.tyBtn2.uiMaskRtStat));
		fUIInRtStatOff(ADR(tyP1031MagSetTeach.tyTeachLifterMag2Slt1Pos.tyBtn2.uiMaskRtStat));
		fUIInRtStatOff(ADR(tyP1031MagSetTeach.tyTeachLifterMag3Slt1Pos.tyBtn2.uiMaskRtStat));

	ELSIF tyP1031MagSetTeach.tyMotionStdLifter.tyBtnJogUp.bRtCompl = TRUE OR tyP1031MagSetTeach.tyMotionStdLifter.tyBtnJogUp.bValue = TRUE THEN
		fUIInRtStatOff(ADR(tyP1031MagSetTeach.tyMotionStdLifter.tyBtnOrigin.uiMaskRtStat));
		fUIInRtStatOff(ADR(tyP1031MagSetTeach.tyMotionStdLifter.tyBtnMovAbs.uiMaskRtStat));
		fUIInRtStatOff(ADR(tyP1031MagSetTeach.tyMotionStdLifter.tyBtnMovRel.uiMaskRtStat));
		fUIInRtStatOff(ADR(tyP1031MagSetTeach.tyMotionStdLifter.tyBtnJogDown.uiMaskRtStat));

		fUIInRtStatOff(ADR(tyP1031MagSetTeach.tyTeachLifterMag1Slt1Pos.tyBtn2.uiMaskRtStat));
		fUIInRtStatOff(ADR(tyP1031MagSetTeach.tyTeachLifterMag2Slt1Pos.tyBtn2.uiMaskRtStat));
		fUIInRtStatOff(ADR(tyP1031MagSetTeach.tyTeachLifterMag3Slt1Pos.tyBtn2.uiMaskRtStat));

	ELSIF tyP1031MagSetTeach.tyTeachLifterMag1Slt1Pos.tyBtn2.bRtCompl = TRUE THEN
		fUIInRtStatOff(ADR(tyP1031MagSetTeach.tyMotionStdLifter.tyBtnOrigin.uiMaskRtStat));
		fUIInRtStatOff(ADR(tyP1031MagSetTeach.tyMotionStdLifter.tyBtnMovAbs.uiMaskRtStat));
		fUIInRtStatOff(ADR(tyP1031MagSetTeach.tyMotionStdLifter.tyBtnMovRel.uiMaskRtStat));
		fUIInRtStatOff(ADR(tyP1031MagSetTeach.tyMotionStdLifter.tyBtnJogUp.uiMaskRtStat));
		fUIInRtStatOff(ADR(tyP1031MagSetTeach.tyMotionStdLifter.tyBtnJogDown.uiMaskRtStat));

	ELSIF tyP1031MagSetTeach.tyTeachLifterMag2Slt1Pos.tyBtn2.bRtCompl = TRUE THEN
		fUIInRtStatOff(ADR(tyP1031MagSetTeach.tyMotionStdLifter.tyBtnOrigin.uiMaskRtStat));
		fUIInRtStatOff(ADR(tyP1031MagSetTeach.tyMotionStdLifter.tyBtnMovAbs.uiMaskRtStat));
		fUIInRtStatOff(ADR(tyP1031MagSetTeach.tyMotionStdLifter.tyBtnMovRel.uiMaskRtStat));
		fUIInRtStatOff(ADR(tyP1031MagSetTeach.tyMotionStdLifter.tyBtnJogUp.uiMaskRtStat));
		fUIInRtStatOff(ADR(tyP1031MagSetTeach.tyMotionStdLifter.tyBtnJogDown.uiMaskRtStat));

	ELSIF tyP1031MagSetTeach.tyTeachLifterMag3Slt1Pos.tyBtn2.bRtCompl = TRUE THEN
		fUIInRtStatOff(ADR(tyP1031MagSetTeach.tyMotionStdLifter.tyBtnOrigin.uiMaskRtStat));
		fUIInRtStatOff(ADR(tyP1031MagSetTeach.tyMotionStdLifter.tyBtnMovAbs.uiMaskRtStat));
		fUIInRtStatOff(ADR(tyP1031MagSetTeach.tyMotionStdLifter.tyBtnMovRel.uiMaskRtStat));
		fUIInRtStatOff(ADR(tyP1031MagSetTeach.tyMotionStdLifter.tyBtnJogUp.uiMaskRtStat));
		fUIInRtStatOff(ADR(tyP1031MagSetTeach.tyMotionStdLifter.tyBtnJogDown.uiMaskRtStat));

	END_IF

	//Axis Error
	IF tyP1031MagSetTeach.tyMotionStdLifter.tyBtnPwr.bRtCompl = TRUE THEN
		fUIInRtStatOff(ADR(tyP1031MagSetTeach.tyMotionStdLifter.tyBtnRst.uiMaskRtStat));
	ELSE
		fUIInRtStatHide(ADR(tyP1031MagSetTeach.tyMotionStdLifter.tyBtnRst.uiMaskRtStat));
	END_IF

	//Interlock Button Get
	IF p_bLifter2AxisErr = TRUE OR p_bLifter2IsHomed = FALSE OR p_bLifter2FwdLmtSen = TRUE OR p_bLifter2RevLmtSen = TRUE THEN
		fUIInRtStatOff(ADR(tyP1031MagSetTeach.tyTeachLifterMag1Slt1Pos.tyBtn1.uiMaskRtStat));
		fUIInRtStatOff(ADR(tyP1031MagSetTeach.tyTeachLifterMag2Slt1Pos.tyBtn1.uiMaskRtStat));
		fUIInRtStatOff(ADR(tyP1031MagSetTeach.tyTeachLifterMag3Slt1Pos.tyBtn1.uiMaskRtStat));
	ELSE
		fUIInRtStatHide(ADR(tyP1031MagSetTeach.tyTeachLifterMag1Slt1Pos.tyBtn1.uiMaskRtStat));
		fUIInRtStatHide(ADR(tyP1031MagSetTeach.tyTeachLifterMag2Slt1Pos.tyBtn1.uiMaskRtStat));
		fUIInRtStatHide(ADR(tyP1031MagSetTeach.tyTeachLifterMag3Slt1Pos.tyBtn1.uiMaskRtStat));
	END_IF

END_ACTION
```

#### Act_OptP1031Lifter2UpdtDat.st
```iecst
ACTION Act_OptP1031Lifter2UpdtDat:

	tyP1031MagSetTeach.tyMotionStdLifter.tyNumCurrPos.diValue		:= p_diLifter2ActualPos;
	tyP1031MagSetTeach.tyMotionStdLifter.tyNumErrCode.diValue		:= UDINT_TO_DINT(p_udiLifter2AxisErrID);
	tyP1031MagSetTeach.tyMotionStdLifter.tyBitmapPwr.usiValueIdx	:= BOOL_TO_USINT(p_bLifter2PwrOn);
	tyP1031MagSetTeach.tyMotionStdLifter.tyBitmapRst.usiValueIdx	:= BOOL_TO_USINT(NOT p_bLifter2AxisErr);
	tyP1031MagSetTeach.tyMotionStdLifter.tyBitmapOrigin.usiValueIdx	:= BOOL_TO_USINT(p_bLifter2IsHomed);
	tyP1031MagSetTeach.tyMotionStdLifter.tyBtnUpLmtSen.bValue		:= p_bLifter2UpSen;
	tyP1031MagSetTeach.tyMotionStdLifter.tyBtnDownLmtSen.bValue		:= p_bLifter2DownSen;

	//Machine Bitmap
	IF p_bLifter2IsHomed = TRUE THEN
		IF p_diLifter2ActualPos <= (p_tyNtParamCurr.tyUILifterTargetPos.diMax / 3) THEN
			tyP1031MagSetTeach.tyMotionStdLifter.tyBitmapMc.uiValueIdx := 2;
		ELSIF p_diLifter2ActualPos <= (p_tyNtParamCurr.tyUILifterTargetPos.diMax / 3 * 2) THEN
			tyP1031MagSetTeach.tyMotionStdLifter.tyBitmapMc.uiValueIdx := 3;
		ELSE
			tyP1031MagSetTeach.tyMotionStdLifter.tyBitmapMc.uiValueIdx := 4;
		END_IF
	ELSE
		tyP1031MagSetTeach.tyMotionStdLifter.tyBitmapMc.uiValueIdx	:= 2;
	END_IF

	IF p_tyNtParamCurr.eProjMag = ULMagDual THEN
		IF p_tyNtParamCurr.bProjLifterMagPlatform AND p_tyNtParamCurr.bUIConvDirRL THEN
			IF 	tyP1031MagSetTeach.tyMotionStdLifter.tyBitmapMc.uiValueIdx < 700 THEN
				tyP1031MagSetTeach.tyMotionStdLifter.tyBitmapMc.uiValueIdx	:= tyP1031MagSetTeach.tyMotionStdLifter.tyBitmapMc.uiValueIdx + 700;
			END_IF
		ELSIF p_tyNtParamCurr.bProjLifterMagPlatform THEN
			IF p_tyNtParamCurr.bProjMagConvLane2Prep = FALSE THEN
				IF 	tyP1031MagSetTeach.tyMotionStdLifter.tyBitmapMc.uiValueIdx < 600 THEN
					tyP1031MagSetTeach.tyMotionStdLifter.tyBitmapMc.uiValueIdx	:= tyP1031MagSetTeach.tyMotionStdLifter.tyBitmapMc.uiValueIdx + 600;
				END_IF
			ELSE
				IF 	tyP1031MagSetTeach.tyMotionStdLifter.tyBitmapMc.uiValueIdx < 903 THEN
					tyP1031MagSetTeach.tyMotionStdLifter.tyBitmapMc.uiValueIdx	:= tyP1031MagSetTeach.tyMotionStdLifter.tyBitmapMc.uiValueIdx + 903;
				END_IF
			END_IF
		ELSIF p_tyNtParamCurr.bMagAutoVerifyPrep = FALSE THEN
			IF 	tyP1031MagSetTeach.tyMotionStdLifter.tyBitmapMc.uiValueIdx < 100 THEN
				tyP1031MagSetTeach.tyMotionStdLifter.tyBitmapMc.uiValueIdx	:= tyP1031MagSetTeach.tyMotionStdLifter.tyBitmapMc.uiValueIdx + 300;
			END_IF
		ELSE
			IF 	tyP1031MagSetTeach.tyMotionStdLifter.tyBitmapMc.uiValueIdx < 300 THEN
				tyP1031MagSetTeach.tyMotionStdLifter.tyBitmapMc.uiValueIdx	:= tyP1031MagSetTeach.tyMotionStdLifter.tyBitmapMc.uiValueIdx + 300;
			END_IF
		END_IF
	ELSIF p_tyNtParamCurr.eProjMag = ULMagTriple AND p_tyNtParamCurr.bProjLifterMagPlatform THEN
		IF p_tyNtParamCurr.bProjLifterMagPlatform AND p_tyNtParamCurr.bUIConvDirRL THEN
			IF 	tyP1031MagSetTeach.tyMotionStdLifter.tyBitmapMc.uiValueIdx < 800 THEN
				tyP1031MagSetTeach.tyMotionStdLifter.tyBitmapMc.uiValueIdx	:= tyP1031MagSetTeach.tyMotionStdLifter.tyBitmapMc.uiValueIdx + 800;
			END_IF
		ELSIF p_tyNtParamCurr.bProjLifterMagPlatform THEN
			IF 	tyP1031MagSetTeach.tyMotionStdLifter.tyBitmapMc.uiValueIdx < 500 THEN
				tyP1031MagSetTeach.tyMotionStdLifter.tyBitmapMc.uiValueIdx	:= tyP1031MagSetTeach.tyMotionStdLifter.tyBitmapMc.uiValueIdx + 500;
			END_IF
		ELSIF p_tyNtParamCurr.bMagAutoVerifyPrep = TRUE AND p_tyNtParamCurr.bProjMotorizedPusherPrep = FALSE THEN
			IF 	tyP1031MagSetTeach.tyMotionStdLifter.tyBitmapMc.uiValueIdx < 200 THEN
				tyP1031MagSetTeach.tyMotionStdLifter.tyBitmapMc.uiValueIdx	:= tyP1031MagSetTeach.tyMotionStdLifter.tyBitmapMc.uiValueIdx + 200;
			END_IF
		ELSIF p_tyNtParamCurr.bMagAutoVerifyPrep = FALSE AND p_tyNtParamCurr.bProjMotorizedPusherPrep = TRUE THEN
			IF 	tyP1031MagSetTeach.tyMotionStdLifter.tyBitmapMc.uiValueIdx < 400 THEN
				tyP1031MagSetTeach.tyMotionStdLifter.tyBitmapMc.uiValueIdx	:= tyP1031MagSetTeach.tyMotionStdLifter.tyBitmapMc.uiValueIdx + 400;
			END_IF
		END_IF
	END_IF

END_ACTION
```

#### Act_OptP1031LifterKeypad.st
```iecst
ACTION Act_OptP1031LifterKeypad:

	IF fUIOutRtStatTPIsOpen(ADR(tyP1031MagSetTeach.tyMotionStdLifter.tyNumTargetPos.uiRtStat)) = TRUE THEN
		tyProperty.tyKeypad.tyStringTitle.sKeypadTitle		:= tyP1031MagSetTeach.tyMotionStdLifter.tyNumTargetPos.sKeypadTitle;

	ELSIF fUIOutRtStatTPIsOpen(ADR(tyP1026McSetTeach.tyMotionStdLifter.tyNumStepSize.uiRtStat)) = TRUE THEN
		tyProperty.tyKeypad.tyStringTitle.sKeypadTitle		:= tyP1031MagSetTeach.tyMotionStdLifter.tyNumStepSize.sKeypadTitle;

	ELSIF fUIOutRtStatTPIsOpen(ADR(tyP1031MagSetTeach.tyMotionStdLifter.tyNumNomSpd.uiRtStat)) = TRUE THEN
		tyProperty.tyKeypad.tyStringTitle.sKeypadTitle		:= tyP1031MagSetTeach.tyMotionStdLifter.tyNumNomSpd.sKeypadTitle;

	ELSIF fUIOutRtStatTPIsOpen(ADR(tyP1031MagSetTeach.tyMotionStdLifter.tyNumSlwSpd.uiRtStat)) = TRUE THEN
		tyProperty.tyKeypad.tyStringTitle.sKeypadTitle		:= tyP1031MagSetTeach.tyMotionStdLifter.tyNumSlwSpd.sKeypadTitle;

	ELSIF fUIOutRtStatTPIsOpen(ADR(tyP1031MagSetTeach.tyTeachLifterMag1Slt1Pos.tyNumNewSlt.uiRtStat)) = TRUE THEN
		tyProperty.tyKeypad.tyStringTitle.sKeypadTitle		:= tyP1031MagSetTeach.tyTeachLifterMag1Slt1Pos.tyNumNewSlt.sKeypadTitle;

	ELSIF fUIOutRtStatTPIsOpen(ADR(tyP1031MagSetTeach.tyTeachLifterMag2Slt1Pos.tyNumNewSlt.uiRtStat)) = TRUE THEN
		tyProperty.tyKeypad.tyStringTitle.sKeypadTitle		:= tyP1031MagSetTeach.tyTeachLifterMag2Slt1Pos.tyNumNewSlt.sKeypadTitle;

	ELSIF fUIOutRtStatTPIsOpen(ADR(tyP1031MagSetTeach.tyTeachLifterMag3Slt1Pos.tyNumNewSlt.uiRtStat)) = TRUE THEN
		tyProperty.tyKeypad.tyStringTitle.sKeypadTitle		:= tyP1031MagSetTeach.tyTeachLifterMag3Slt1Pos.tyNumNewSlt.sKeypadTitle;

//	ELSIF fUIOutRtStatTPIsOpen(ADR(tyP1031MagSetTeach.tyTeachLifterMag4Slt1Pos.tyNumNewSlt.uiRtStat)) = TRUE THEN
//		tyProperty.tyKeypad.tyStringTitle.sKeypadTitle		:= tyP1031MagSetTeach.tyTeachLifterMag4Slt1Pos.tyNumNewSlt.sKeypadTitle;
//
	END_IF

END_ACTION
```

#### Act_OptP1031LifterRstMnl.st
```iecst
ACTION Act_OptP1031LifterRstMnl:

	IF EDGEPOS((bManualMod = FALSE) OR (p_eLifterBtmStatus = Error)) THEN

		bJogSlow				:= FALSE;
		bJogFast				:= FALSE;
		fbJogSlowToFastDlyTm.IN	:= FALSE;

		tyP1031MagSetTeach.tyMotionStdLifter.tyBtnPwr.bRtCompl			:= FALSE;
		tyP1031MagSetTeach.tyMotionStdLifter.tyBtnStop.bRtCompl			:= FALSE;
		tyP1031MagSetTeach.tyMotionStdLifter.tyBtnOrigin.bRtCompl		:= FALSE;
		tyP1031MagSetTeach.tyMotionStdLifter.tyBtnRst.bRtCompl			:= FALSE;
		tyP1031MagSetTeach.tyMotionStdLifter.tyBtnMovAbs.bRtCompl		:= FALSE;
		tyP1031MagSetTeach.tyMotionStdLifter.tyBtnMovRel.bRtCompl		:= FALSE;
		tyP1031MagSetTeach.tyMotionStdLifter.tyBtnJogUp.bRtCompl		:= FALSE;
		tyP1031MagSetTeach.tyMotionStdLifter.tyBtnJogDown.bRtCompl		:= FALSE;

		tyP1031MagSetTeach.tyTeachLifterMag1Slt1Pos.tyBtn2.bRtCompl		:= FALSE;
		tyP1031MagSetTeach.tyTeachLifterMag2Slt1Pos.tyBtn2.bRtCompl		:= FALSE;
		tyP1031MagSetTeach.tyTeachLifterMag3Slt1Pos.tyBtn2.bRtCompl		:= FALSE;

		tyP1031MagSetTeach.tyMotionStdLifter.tyBtnPwr.bValue			:= FALSE;
		tyP1031MagSetTeach.tyMotionStdLifter.tyBtnStop.bValue			:= TRUE;
		tyP1031MagSetTeach.tyMotionStdLifter.tyBtnOrigin.bValue			:= FALSE;
		tyP1031MagSetTeach.tyMotionStdLifter.tyBtnRst.bValue			:= FALSE;
		tyP1031MagSetTeach.tyMotionStdLifter.tyBtnMovAbs.bValue			:= FALSE;
		tyP1031MagSetTeach.tyMotionStdLifter.tyBtnMovRel.bValue			:= FALSE;
		tyP1031MagSetTeach.tyMotionStdLifter.tyBtnJogUp.bValue			:= FALSE;
		tyP1031MagSetTeach.tyMotionStdLifter.tyBtnJogDown.bValue		:= FALSE;

		tyP1031MagSetTeach.tyTeachLifterMag1Slt1Pos.tyBtn2.bValue		:= FALSE;
		tyP1031MagSetTeach.tyTeachLifterMag2Slt1Pos.tyBtn2.bValue		:= FALSE;
		tyP1031MagSetTeach.tyTeachLifterMag3Slt1Pos.tyBtn2.bValue		:= FALSE;

		tyP1031MagSetTeach.tyMotionStdLifter.tyBtnPwr.bRtLk				:= FALSE;
		tyP1031MagSetTeach.tyMotionStdLifter.tyBtnStop.bRtLk			:= TRUE;
		tyP1031MagSetTeach.tyMotionStdLifter.tyBtnOrigin.bRtLk			:= FALSE;
		tyP1031MagSetTeach.tyMotionStdLifter.tyBtnRst.bRtLk				:= FALSE;
		tyP1031MagSetTeach.tyMotionStdLifter.tyBtnMovAbs.bRtLk			:= FALSE;
		tyP1031MagSetTeach.tyMotionStdLifter.tyBtnMovRel.bRtLk			:= FALSE;
		tyP1031MagSetTeach.tyMotionStdLifter.tyBtnJogUp.bRtLk			:= FALSE;
		tyP1031MagSetTeach.tyMotionStdLifter.tyBtnJogDown.bRtLk			:= FALSE;

		tyP1031MagSetTeach.tyTeachLifterMag1Slt1Pos.tyBtn2.bRtLk		:= FALSE;
		tyP1031MagSetTeach.tyTeachLifterMag2Slt1Pos.tyBtn2.bRtLk		:= FALSE;
		tyP1031MagSetTeach.tyTeachLifterMag3Slt1Pos.tyBtn2.bRtLk		:= FALSE;

		tyP1031MagSetTeach.tyMotionStdLifter.tyBtnPwr.uiMaskRtStat		:= TRUE;
		tyP1031MagSetTeach.tyMotionStdLifter.tyBtnOrigin.uiMaskRtStat	:= FALSE;
		tyP1031MagSetTeach.tyMotionStdLifter.tyBtnRst.uiMaskRtStat		:= TRUE;
		tyP1031MagSetTeach.tyMotionStdLifter.tyBtnMovAbs.uiMaskRtStat	:= FALSE;
		tyP1031MagSetTeach.tyMotionStdLifter.tyBtnMovRel.uiMaskRtStat	:= FALSE;
		tyP1031MagSetTeach.tyMotionStdLifter.tyBtnJogUp.uiMaskRtStat	:= FALSE;
		tyP1031MagSetTeach.tyMotionStdLifter.tyBtnJogDown.uiMaskRtStat	:= FALSE;

		tyP1031MagSetTeach.tyTeachLifterMag1Slt1Pos.tyBtn2.uiMaskRtStat	:= FALSE;
		tyP1031MagSetTeach.tyTeachLifterMag2Slt1Pos.tyBtn2.uiMaskRtStat	:= FALSE;
		tyP1031MagSetTeach.tyTeachLifterMag3Slt1Pos.tyBtn2.uiMaskRtStat	:= FALSE;

		eInShutterAct	:= PneuActIdle;
		eOutShutterAct	:= PneuActIdle;
		eOutShutterAct2	:= PneuActIdle;
		eOutShutterAct3	:= PneuActIdle;
		eLifterBtmAct	:= LifterActIdle;

		tyP1031MagSetTeach.tyInOutletShutterFB.tyBtnClose.bRtCompl	:= FALSE;
		tyP1031MagSetTeach.tyInOutletShutterFB.tyBtnClose.bValue	:= FALSE;
		tyP1031MagSetTeach.tyInOutletShutterFB.tyBtnOpen.bRtCompl	:= FALSE;
		tyP1031MagSetTeach.tyInOutletShutterFB.tyBtnOpen.bValue	:= FALSE;

	END_IF

END_ACTION
```

#### Act_EntP1040Disp.st
```iecst
ACTION Act_EntP1040Disp:

	//Access Address
	p_tyC0005Main ACCESS ADR(tyCommon.tyMain);

	p_tyC0007Notif ACCESS ADR(tyCommon.tyNotif);

	p_tyC0008MsgBox ACCESS ADR(tyP1040ProdSet.tyMsgBoxHide);

	p_tyC0009Info ACCESS ADR(tyCommon.tyInfo);

	p_tyC0011RcpPopUp ACCESS ADR(tyP1040ProdSet.tyRcpPopUp);

	p_tyP1040ProdSet ACCESS ADR(tyP1040ProdSet.tyProdSet);

	//Display
	udiP1040SelectedRowOld	 := 0;

	tyP1040ProdSet.tyProdSet.tyBtnLongBrd.uiRtStat.0		:= NOT(p_tyNtParamCurr.bProjLongBrdPrep AND p_tyMcParamCurr.bLongBrdEn);

	tyP1040ProdSet.tyProdSet.tyBtnGapBetBrds.uiRtStat.0		:= NOT p_tyMcParamCurr.bGapBwtnBrdEn;

	tyP1040ProdSet.tyProdSet.tyNumMinReqFreeBffr.diValueMax	:= p_tyMagRcpCurrRcp.diTtlSlt;
	tyP1040ProdSet.tyProdSet.tyNumLastSlt.diValueMax		:= p_tyMagRcpCurrRcp.diTtlSlt;

	fUIInRtStatHide(ADR(tyP1040ProdSet.tyRcpPopUp.tyLyr.uiRtStat));

	tyP1040ProdSet.tyProdSet.tyBtnSort.bValue := FALSE;
	tyP1040ProdSet.tyProdSet.tyBtnSort.bRtCompl := FALSE;

END_ACTION
```

#### Act_OptP1040Mask.st
```iecst
ACTION Act_OptP1040Mask:

	IF tyP1040ProdSet.tyProdSet.tyNumProdWidth.bRtCompl 			OR tyP1040ProdSet.tyProdSet.tyStringRecipeNm.bRtCompl
		OR tyP1040ProdSet.tyProdSet.tyDrpDnMcMode.bRtCompl			OR tyP1040ProdSet.tyProdSet.tyNumFirstSlt.bRtCompl
		OR tyP1040ProdSet.tyProdSet.tyNumLastSlt.bRtCompl			OR tyP1040ProdSet.tyProdSet.tyNumPitch.bRtCompl
		OR tyP1040ProdSet.tyProdSet.tyBtnToptoBtm.bRtCompl			OR tyP1040ProdSet.tyProdSet.tyBtnLongBrd.bRtCompl
		OR tyP1040ProdSet.tyProdSet.tyBtnGapBetBrds.bRtCompl		OR tyP1040ProdSet.tyProdSet.tyNumBrdPerSlt.bRtCompl
		OR tyP1040ProdSet.tyProdSet.tyNumMinReqFreeBffr.bRtCompl	OR tyP1040ProdSet.tyProdSet.tyNumProdWidth2.bRtCompl
		OR tyP1040ProdSet.tyProdSet.tyNumMtrPshrExtSpd.bRtCompl 	OR tyP1040ProdSet.tyProdSet.tyNumMtrPshrExtTorq.bRtCompl
		OR tyP1040ProdSet.tyProdSet.tyNumPshrOffset.bRtCompl
		THEN

		fUIInRtStatHide(ADR(tyP1040ProdSet.tyProdSet.tyBtnSave.uiMaskRtStat));

		tyP1040ProdSet.tyProdSet.tyNumProdWidth.bRtCompl		:= FALSE;
		tyP1040ProdSet.tyProdSet.tyNumProdWidth2.bRtCompl		:= FALSE;
		tyP1040ProdSet.tyProdSet.tyStringRecipeNm.bRtCompl		:= FALSE;
		tyP1040ProdSet.tyProdSet.tyNumFirstSlt.bRtCompl			:= FALSE;
		tyP1040ProdSet.tyProdSet.tyNumLastSlt.bRtCompl			:= FALSE;
		tyP1040ProdSet.tyProdSet.tyNumPitch.bRtCompl			:= FALSE;
		tyP1040ProdSet.tyProdSet.tyBtnToptoBtm.bRtCompl			:= FALSE;
		tyP1040ProdSet.tyProdSet.tyBtnLongBrd.bRtCompl			:= FALSE;
		tyP1040ProdSet.tyProdSet.tyBtnGapBetBrds.bRtCompl		:= FALSE;
		tyP1040ProdSet.tyProdSet.tyNumBrdPerSlt.bRtCompl		:= FALSE;
		tyP1040ProdSet.tyProdSet.tyDrpDnMcMode.bRtCompl			:= FALSE;
		tyP1040ProdSet.tyProdSet.tyNumMinReqFreeBffr.bRtCompl	:= FALSE;
		tyP1040ProdSet.tyProdSet.tyNumMtrPshrExtSpd.bRtCompl	:= FALSE;
		tyP1040ProdSet.tyProdSet.tyNumMtrPshrExtTorq.bRtCompl	:= FALSE;
		tyP1040ProdSet.tyProdSet.tyNumPshrOffset.bRtCompl		:= FALSE;
	END_IF

	IF (tyP1040ProdSet.tyProdSet.tyTableRecipe.a_tyStringDataCol1[tyP1040Table.uiSelectedRow].sValue <> '') AND (tyP1040ProdSet.tyProdSet.tyBtnSave.bRtCompl = FALSE) AND (tyP1040ProdSet.tyProdSet.tyBtnToXML.bRtCompl = FALSE) AND (tyP1040ProdSet.tyProdSet.tyBtnFromXML.bRtCompl = FALSE) THEN
		fUIInRtStatHide(ADR(tyP1040ProdSet.tyProdSet.tyBtnDelete.uiMaskRtStat));
	ELSE
		fUIInRtStatOff(ADR(tyP1040ProdSet.tyProdSet.tyBtnDelete.uiMaskRtStat));
	END_IF

	tyP1040ProdSet.tyProdSet.tyBtnToXML.uiMaskRtStat.0		:= (tyP1040ProdSet.tyProdSet.tyBtnSave.uiMaskRtStat.0 = FALSE) AND (tyP1040ProdSet.tyProdSet.tyBtnDelete.bRtCompl = FALSE) AND (tyP1040ProdSet.tyProdSet.tyBtnFromXML.bRtCompl = FALSE);
	tyP1040ProdSet.tyProdSet.tyBtnFromXML.uiMaskRtStat.0	:= (tyP1040ProdSet.tyProdSet.tyBtnSave.uiMaskRtStat.0 = FALSE) AND (tyP1040ProdSet.tyProdSet.tyBtnDelete.bRtCompl = FALSE) AND (tyP1040ProdSet.tyProdSet.tyBtnToXML.bRtCompl = FALSE);

	tyP1040ProdSet.tyProdSet.tyBtnSort.uiMaskRtStat.0		:= (tyP1040ProdSet.tyProdSet.tyTableRecipe.a_tyStringDataCol1[1].sValue <> '') AND (tyP1040ProdSet.tyProdSet.tyStringSearch.bRtCompl = FALSE)
																AND (tyP1040ProdSet.tyProdSet.tyBtnSave.uiMaskRtStat.0 = FALSE) AND (tyP1040ProdSet.tyProdSet.tyBtnDelete.bRtCompl = FALSE)
																AND (tyP1040ProdSet.tyProdSet.tyBtnToXML.bRtCompl = FALSE) AND (tyP1040ProdSet.tyProdSet.tyBtnFromXML.bRtCompl = FALSE);

END_ACTION
```
